# B&R Automation Studio project Panasonic_LinkaPowerCP2_A2021055 (part 45)

#### Main.st - Init, cyclic, exit code
```iecst
PROGRAM _INIT
	(* Insert code here *)
	SKTcpClientTrace_1.Params.IPportClient := 22000;
	SKTcpClientTrace_1.Cmd.LoggerOn:= FALSE;
END_PROGRAM

PROGRAM _CYCLIC

	//Priradenie indexu paletky//
    a:= P4_Etiketovacka.PAR.CisloPaletky;
	P4_Etiketovacka.PAR.CisloPaletky_STRING:= USINT_TO_STRING(a);

    //Parametre komunikácie//
    memcpy(ADR(SKTcpClientTrace_1.Params.IPaddrServ),ADR('192.168.128.250'),SIZEOF('192.168.128.250'));

    SKTcpClientTrace_1.Params.IPportServ := 12000;

	SKTcpClientTrace_1.pDevice := ADR('HDD_LOGGER');
	SKTcpClientTrace_1.pFile := ADR('logger_sktcpclienttrace_9.log');
    SKTcpClientTrace_1();

    //Parametre komunikácie//
    //Vstupy pre server//
    SKTcpClientTrace_1.Params.Packet.type := TRCB_P4_Etiketovacka_ST9.INPUTS.TYP_Prikazu;
    SKTcpClientTrace_1.Params.Packet.workplace := TRCB_P4_Etiketovacka_ST9.INPUTS.CisloStanice;
    SKTcpClientTrace_1.Params.Packet.rfid := TRCB_P4_Etiketovacka_ST9.INPUTS.CisloPaletky;
    SKTcpClientTrace_1.Params.Packet.master := TRCB_P4_Etiketovacka_ST9.INPUTS.QRkodPowerCP;
    SKTcpClientTrace_1.Params.Packet.dps1:= TRCB_P4_Etiketovacka_ST9.INPUTS.QRkodFiltra;
    SKTcpClientTrace_1.Params.Packet.dps2:= '';
    SKTcpClientTrace_1.Params.Packet.dps3:= '';
    SKTcpClientTrace_1.Params.Packet.dps4:= '';
    SKTcpClientTrace_1.Params.Packet.dps5:= '';
    SKTcpClientTrace_1.Params.Packet.operator_id := TRCB_P4_Etiketovacka_ST9.INPUTS.ID_Operatora;
    SKTcpClientTrace_1.Params.Packet.data_report:= TRCB_P4_Etiketovacka_ST9.INPUTS.Report;
    SKTcpClientTrace_1.Params.Packet.result := TRCB_P4_Etiketovacka_ST9.INPUTS.StavPaletky;

    //Výstupy zo servera//
    TRCB_P4_Etiketovacka_ST9.OUTPUTS.TYP_Prikazu:= SKTcpClientTrace_1.Internal.Splitter.out[1];
    TRCB_P4_Etiketovacka_ST9.OUTPUTS.CisloStanice:= SKTcpClientTrace_1.Internal.Splitter.out[2];
    TRCB_P4_Etiketovacka_ST9.OUTPUTS.CisloPaletky:= SKTcpClientTrace_1.Internal.Splitter.out[3];
    IF TRCB_P4_Etiketovacka_ST9.INPUTS.TYP_Prikazu = '0' THEN
        TRCB_P4_Etiketovacka_ST9.OUTPUTS.CisloEtikety:= SKTcpClientTrace_1.Internal.Splitter.out[4];
    ELSE
        TRCB_P4_Etiketovacka_ST9.OUTPUTS.QRkodPowerCP:= SKTcpClientTrace_1.Internal.Splitter.out[4];
    END_IF
    TRCB_P4_Etiketovacka_ST9.OUTPUTS.QRkodFiltra:= SKTcpClientTrace_1.Internal.Splitter.out[5];
    TRCB_P4_Etiketovacka_ST9.OUTPUTS.ID_Operatora:= SKTcpClientTrace_1.Internal.Splitter.out[10];
    TRCB_P4_Etiketovacka_ST9.OUTPUTS.DruhCinnostiNaPaletke:= SKTcpClientTrace_1.Internal.Splitter.out[11];
    TRCB_P4_Etiketovacka_ST9.OUTPUTS.PovolenieCinnostiNaPaletke:= SKTcpClientTrace_1.Internal.Splitter.out[12];

    //Volanie funkcie SequenceControl//
    SequenceControl(SC:= SC_KOM_Server);

    CASE SC_KOM_Server.Step OF

        0:
            SC_KOM_Server.StepName:= '0 - Nulovanie';
            SKTcpClientTrace_1.Cmd.Send:= FALSE;
            TRCB_P4_Etiketovacka_ST9.CMD.VyziadajStavPaletky_TYP1:= FALSE;
            TRCB_P4_Etiketovacka_ST9.CMD.PriradQRkodFiltra_TYP3:= FALSE;
            TRCB_P4_Etiketovacka_ST9.CMD.VyziadajCisloEtikety_TYP0:= FALSE;
			TRCB_P4_Etiketovacka_ST9.CMD.OdosliStavPaletky_TYP2:= FALSE;
			TRCB_P4_Etiketovacka_ST9.CMD.VyziadajStavPanatrace_TYP4:= FALSE;
            TRCB_P4_Etiketovacka_ST9.STATUS.KomunikaciaUkoncena:= FALSE;
			TRCB_P4_Etiketovacka_ST9.STATUS.KomunikaciaError:= FALSE;
			TRCB_P4_Etiketovacka_ST9.STATUS.KOM_READY:= FALSE;
            PocetDopytovNaServer:= 0;

            IF SKTcpClientTrace_1.Internal.Step = 0 THEN
                SKTcpClientTrace_1.Enable:= TRUE;
                SC_KOM_Server.ResetStep:= TRUE;
                SC_KOM_Server.Step:= 1;
            ELSIF SKTcpClientTrace_1.Internal.Step = 15 THEN
                SKTcpClientTrace_1.Enable:= TRUE;
                SC_KOM_Server.ResetStep:= TRUE;
                SC_KOM_Server.Step:= 1;
            ELSE
                SKTcpClientTrace_1.Enable:= FALSE;
            END_IF

        1:
            SC_KOM_Server.StepName:= '1 - Rozhodnutie o cinnosti';
            TRCB_P4_Etiketovacka_ST9.STATUS.KOM_READY:= TRUE;
			IF TRCB_P4_Etiketovacka_ST9.CMD.VyziadajStavPaletky_TYP1 THEN
                TRCB_P4_Etiketovacka_ST9.STATUS.KOM_READY:= FALSE;
				SC_KOM_Server.Step:= 10;
            ELSIF TRCB_P4_Etiketovacka_ST9.CMD.PriradQRkodFiltra_TYP3 THEN
                TRCB_P4_Etiketovacka_ST9.STATUS.KOM_READY:= FALSE;
				SC_KOM_Server.Step:= 20;
            ELSIF TRCB_P4_Etiketovacka_ST9.CMD.VyziadajCisloEtikety_TYP0 THEN
                TRCB_P4_Etiketovacka_ST9.STATUS.KOM_READY:= FALSE;
				SC_KOM_Server.Step:= 30;
            ELSIF TRCB_P4_Etiketovacka_ST9.CMD.OdosliStavPaletky_TYP2 THEN
				TRCB_P4_Etiketovacka_ST9.STATUS.KOM_READY:= FALSE;
				SC_KOM_Server.Step:= 40;
			ELSIF TRCB_P4_Etiketovacka_ST9.CMD.VyziadajStavPanatrace_TYP4 THEN
				TRCB_P4_Etiketovacka_ST9.STATUS.KOM_READY:= FALSE;
				SC_KOM_Server.Step:= 50;
            END_IF

        10:
            SC_KOM_Server.StepName:= '10 - Vyziadanie stavu paletky - odoslanie dat na server';
            SC_KOM_Server.IdleTime.PT:= T#3s;
            SC_KOM_Server.AlarmTime.PT:= T#10s;
            SC_KOM_Server.AlarmTime.IN:= TRUE;

			TRCB_P4_Etiketovacka_ST9.INPUTS.CisloPaletky:= 'Pal';
			brsstrcat(ADR(TRCB_P4_Etiketovacka_ST9.INPUTS.CisloPaletky), ADR(P4_Etiketovacka.PAR.CisloPaletky_STRING));

            TRCB_P4_Etiketovacka_ST9.INPUTS.TYP_Prikazu:= '1';
            TRCB_P4_Etiketovacka_ST9.INPUTS.CisloStanice:= 'ST9';
            TRCB_P4_Etiketovacka_ST9.INPUTS.QRkodPowerCP:= Paletka[a].PAR.QRkodPowerCP;
            TRCB_P4_Etiketovacka_ST9.INPUTS.QRkodFiltra:= '';
            TRCB_P4_Etiketovacka_ST9.INPUTS.ID_Operatora:= Paletka[a].PAR.ID_Operatora;
            TRCB_P4_Etiketovacka_ST9.INPUTS.Report:= '';
            TRCB_P4_Etiketovacka_ST9.INPUTS.StavPaletky:= 'OK';

			IF SKTcpClientTrace_1.Status.staReadyToSend AND NOT SKTcpClientTrace_1.Cmd.Close THEN
				TRCB_P4_Etiketovacka_ST9.OUTPUTS.TYP_Prikazu:= '';
				SKTcpClientTrace_1.Cmd.Send:= TRUE;
				SC_KOM_Server.ResetStep:= TRUE;
				SC_KOM_Server.Step:= 13;
			END_IF

		13:
            SC_KOM_Server.StepName:= '13 - Vyziadanie stavu paletky - odpoved servera';
            SC_KOM_Server.IdleTime.PT:= T#3s;
            SC_KOM_Server.AlarmTime.PT:= T#7s;
            SC_KOM_Server.AlarmTime.IN:= TRUE;

            IF SKTcpClientTrace_1.Status.staReceived AND
                (TRCB_P4_Etiketovacka_ST9.OUTPUTS.TYP_Prikazu = TRCB_P4_Etiketovacka_ST9.INPUTS.TYP_Prikazu) AND
                (TRCB_P4_Etiketovacka_ST9.OUTPUTS.QRkodPowerCP = TRCB_P4_Etiketovacka_ST9.INPUTS.QRkodPowerCP) THEN
                TRCB_P4_Etiketovacka_ST9.STATUS.KomunikaciaUkoncena:= TRUE;
                SC_KOM_Server.ResetStep:= TRUE;
                SC_KOM_Server.Step:= 15;
            ELSIF SC_KOM_Server.AlarmTime.Q AND NOT SKTcpClientTrace_1.Status.staSending THEN
                PocetDopytovNaServer:= PocetDopytovNaServer + 1;
				SKTcpClientTrace_1.Cmd.Send:= FALSE;
				SKTcpClientTrace_1.Cmd.Close:= TRUE;
				SC_KOM_Server.ResetStep:= TRUE;
                SC_KOM_Server.Step:= 14;
            END_IF

        14:
            SC_KOM_Server.StepName:= '14 - Vyziadanie stavu paletky - cakam na opatovny dopyt na server';
            SC_KOM_Server.IdleTime.PT:= T#1s;
            SC_KOM_Server.AlarmTime.PT:= T#10s;
            SC_KOM_Server.IdleTime.IN:= TRUE;

            IF PocetDopytovNaServer < 3 THEN
                IF SC_KOM_Server.IdleTime.Q THEN
                    SC_KOM_Server.ResetStep:= TRUE;
                    SC_KOM_Server.Step:= 10;
                END_IF
            ELSE
                TRCB_P4_Etiketovacka_ST9.STATUS.KomunikaciaError:= TRUE;
                SC_KOM_Server.ResetStep:= TRUE;
                SC_KOM_Server.Step:= 15;
            END_IF

        15:
            SC_KOM_Server.StepName:= '15 - Vyziadanie stavu paletky - cakam na ukoncenie komunikacie';
            SC_KOM_Server.IdleTime.PT:= T#3s;
            SC_KOM_Server.AlarmTime.PT:= T#10s;

            IF NOT TRCB_P4_Etiketovacka_ST9.CMD.VyziadajStavPaletky_TYP1 THEN
                SC_KOM_Server.ResetStep:= TRUE;
                SC_KOM_Server.Step:= 0;
            END_IF

        20:
            SC_KOM_Server.StepName:= '20 - Priradenie QR kodu - odoslanie dat na server';
            SC_KOM_Server.IdleTime.PT:= T#3s;
            SC_KOM_Server.AlarmTime.PT:= T#10s;

            TRCB_P4_Etiketovacka_ST9.INPUTS.TYP_Prikazu:= '3';
            TRCB_P4_Etiketovacka_ST9.INPUTS.CisloStanice:= 'ST9';
            TRCB_P4_Etiketovacka_ST9.INPUTS.CisloPaletky;
            TRCB_P4_Etiketovacka_ST9.INPUTS.QRkodPowerCP:= Paletka[a].PAR.QRkodPowerCP;
            TRCB_P4_Etiketovacka_ST9.INPUTS.QRkodFiltra:= '';
            TRCB_P4_Etiketovacka_ST9.INPUTS.ID_Operatora:= Paletka[a].PAR.ID_Operatora;
            TRCB_P4_Etiketovacka_ST9.INPUTS.Report:= '';
            TRCB_P4_Etiketovacka_ST9.INPUTS.StavPaletky:= 'OK';
            SKTcpClientTrace_1.Cmd.Send:= TRUE;

            IF SKTcpClientTrace_1.Cmd.Send AND NOT SKTcpClientTrace_1.Status.staReceived AND NOT SKTcpClientTrace_1.Status.staError THEN
                SC_KOM_Server.ResetStep:= TRUE;
                SC_KOM_Server.Step:= 23;
            END_IF

        23:
            SC_KOM_Server.StepName:= '23 - Priradenie QR kodu - odpoved servera';
            SC_KOM_Server.IdleTime.PT:= T#3s;
            SC_KOM_Server.AlarmTime.PT:= T#20s;
            SC_KOM_Server.AlarmTime.IN:= TRUE;

            IF SKTcpClientTrace_1.Status.staReceived AND
                (TRCB_P4_Etiketovacka_ST9.OUTPUTS.TYP_Prikazu = TRCB_P4_Etiketovacka_ST9.INPUTS.TYP_Prikazu) AND
                (TRCB_P4_Etiketovacka_ST9.OUTPUTS.QRkodPowerCP = TRCB_P4_Etiketovacka_ST9.INPUTS.QRkodPowerCP) THEN
                TRCB_P4_Etiketovacka_ST9.STATUS.KomunikaciaUkoncena:= TRUE;
                SC_KOM_Server.ResetStep:= TRUE;
                SC_KOM_Server.Step:= 25;
            ELSIF SC_KOM_Server.AlarmTime.Q THEN
                TRCB_P4_Etiketovacka_ST9.STATUS.KomunikaciaError:= TRUE;
                SC_KOM_Server.ResetStep:= TRUE;
                SC_KOM_Server.Step:= 25;
            END_IF

        25:
            SC_KOM_Server.StepName:= '25 - Priradenie QR kodu - cakam na ukoncenie komunikacie';
            SC_KOM_Server.IdleTime.PT:= T#3s;
            SC_KOM_Server.AlarmTime.PT:= T#10s;

            IF NOT TRCB_P4_Etiketovacka_ST9.CMD.PriradQRkodFiltra_TYP3 THEN
                SC_KOM_Server.ResetStep:= TRUE;
                SC_KOM_Server.Step:= 0;
            END_IF

        30:
            SC_KOM_Server.StepName:= '30 - Vyziadanie serioveho cisla - odoslanie dat na server';
            SC_KOM_Server.IdleTime.PT:= T#3s;
            SC_KOM_Server.AlarmTime.PT:= T#20s;
            SC_KOM_Server.AlarmTime.IN:= TRUE;

			TRCB_P4_Etiketovacka_ST9.INPUTS.CisloPaletky:= 'Pal';
			brsstrcat(ADR(TRCB_P4_Etiketovacka_ST9.INPUTS.CisloPaletky), ADR(P4_Etiketovacka.PAR.CisloPaletky_STRING));

            TRCB_P4_Etiketovacka_ST9.INPUTS.TYP_Prikazu:= '0';
            TRCB_P4_Etiketovacka_ST9.INPUTS.CisloStanice:= 'ST9';
            TRCB_P4_Etiketovacka_ST9.INPUTS.QRkodPowerCP:= '';
            TRCB_P4_Etiketovacka_ST9.INPUTS.QRkodFiltra:= '';
            TRCB_P4_Etiketovacka_ST9.INPUTS.ID_Operatora:= Paletka[a].PAR.ID_Operatora;
            TRCB_P4_Etiketovacka_ST9.INPUTS.Report:= '';
            TRCB_P4_Etiketovacka_ST9.INPUTS.StavPaletky:= 'OK';

			IF SKTcpClientTrace_1.Status.staReadyToSend AND NOT SKTcpClientTrace_1.Cmd.Close THEN
				TRCB_P4_Etiketovacka_ST9.OUTPUTS.TYP_Prikazu:= '';
				SKTcpClientTrace_1.Cmd.Send:= TRUE;
				SC_KOM_Server.ResetStep:= TRUE;
				SC_KOM_Server.Step:= 33;
			END_IF

        33:
            SC_KOM_Server.StepName:= '33 - Vyziadanie serioveho cisla - odpoved servera';
			SC_KOM_Server.IdleTime.PT:= T#3s;
            SC_KOM_Server.AlarmTime.PT:= T#7s;
            SC_KOM_Server.AlarmTime.IN:= TRUE;

            IF SKTcpClientTrace_1.Status.staReceived AND
                (TRCB_P4_Etiketovacka_ST9.OUTPUTS.TYP_Prikazu = TRCB_P4_Etiketovacka_ST9.INPUTS.TYP_Prikazu) THEN
                TRCB_P4_Etiketovacka_ST9.STATUS.KomunikaciaUkoncena:= TRUE;
                SC_KOM_Server.ResetStep:= TRUE;
                SC_KOM_Server.Step:= 35;
            ELSIF SC_KOM_Server.AlarmTime.Q AND NOT SKTcpClientTrace_1.Status.staSending THEN
                PocetDopytovNaServer:= PocetDopytovNaServer + 1;
				SKTcpClientTrace_1.Cmd.Send:= FALSE;
				SKTcpClientTrace_1.Cmd.Close:= TRUE;
				SC_KOM_Server.ResetStep:= TRUE;
                SC_KOM_Server.Step:= 34;
            END_IF

        34:
            SC_KOM_Server.StepName:= '34 - Vyziadanie serioveho cisla - cakam na opatovny dopyt na server';
            SC_KOM_Server.IdleTime.PT:= T#1s;
            SC_KOM_Server.AlarmTime.PT:= T#10s;
            SC_KOM_Server.IdleTime.IN:= TRUE;
            SKTcpClientTrace_1.Cmd.Send:= FALSE;

            IF PocetDopytovNaServer < 3 THEN
                IF SC_KOM_Server.IdleTime.Q THEN
                    SC_KOM_Server.ResetStep:= TRUE;
                    SC_KOM_Server.Step:= 30;
                END_IF
            ELSE
                TRCB_P4_Etiketovacka_ST9.STATUS.KomunikaciaError:= TRUE;
                SC_KOM_Server.ResetStep:= TRUE;
                SC_KOM_Server.Step:= 35;
            END_IF

        35:
            SC_KOM_Server.StepName:= '35 - Vyziadanie serioveho cisla - cakam na ukoncenie komunikacie';
            SC_KOM_Server.IdleTime.PT:= T#3s;
            SC_KOM_Server.AlarmTime.PT:= T#10s;

            IF NOT TRCB_P4_Etiketovacka_ST9.CMD.VyziadajCisloEtikety_TYP0 THEN
                SC_KOM_Server.ResetStep:= TRUE;
                SC_KOM_Server.Step:= 0;
            END_IF

        40:
            SC_KOM_Server.StepName:= '40 - Odoslanie stavu paletky - odoslanie dat na server';
            SC_KOM_Server.IdleTime.PT:= T#3s;
            SC_KOM_Server.AlarmTime.PT:= T#20s;
            SC_KOM_Server.AlarmTime.IN:= TRUE;

            IF NOT SC_KOM_Server.Switch1 THEN
                brsmemset(ADR(Report),0,SIZEOF(Report));
               	brsmemset(ADR(TRCB_P4_Etiketovacka_ST9.INPUTS.Report), 0, SIZEOF(TRCB_P4_Etiketovacka_ST9.INPUTS.Report));

				//Kamera 15//
                Report[0].PoradoveCislo:= '1';
                Report[0].Popis:= 'KAM_15_KontrolaEtikety';
                Report[0].FormatHodnoty:= '2';
                Report[0].Tolerancia_MIN_Hodnota:= '';
                Report[0].Tolerancia_MAX_Hodnota:= '';
                Report[0].Nominal:= 'OK';
                Report[0].Tolerancia_MIN_Jednotky:= '';
                Report[0].Tolerancia_MAX_Jednotky:= '';
                IF Reports.Kamery.P4_CAM15_KontrolaPaletky = 'PASS' THEN
                    Report[0].NameranaHodnota:= 'OK';
                ELSE
                    Report[0].NameranaHodnota:= 'NG';
                END_IF
                Report[0].NameranaHodnota_Jednotky:= '';
                Report[0].VyslednyResult:= Reports.Kamery.P4_CAM15_KontrolaPaletky;
                SKTcpClientNewCsvEntry(Report[0].PoradoveCislo,Report[0].Popis,Report[0].FormatHodnoty,Report[0].Tolerancia_MIN_Hodnota,Report[0].Tolerancia_MAX_Hodnota,Report[0].Nominal,Report[0].Tolerancia_MIN_Jednotky,Report[0].Tolerancia_MAX_Jednotky,Report[0].NameranaHodnota,Report[0].NameranaHodnota_Jednotky,Report[0].VyslednyResult, ADR(TRCB_P4_Etiketovacka_ST9.INPUTS.Report));
                SC_KOM_Server.Switch1:= TRUE;
            END_IF

			TRCB_P4_Etiketovacka_ST9.INPUTS.CisloPaletky:= 'Pal';
			brsstrcat(ADR(TRCB_P4_Etiketovacka_ST9.INPUTS.CisloPaletky), ADR(P4_Etiketovacka.PAR.CisloPaletky_STRING));

            TRCB_P4_Etiketovacka_ST9.INPUTS.TYP_Prikazu:= '2';
            TRCB_P4_Etiketovacka_ST9.INPUTS.CisloStanice:= 'ST9';
            TRCB_P4_Etiketovacka_ST9.INPUTS.QRkodPowerCP:= Paletka[a].PAR.QRkodPowerCP;
            TRCB_P4_Etiketovacka_ST9.INPUTS.QRkodFiltra:= '';
            TRCB_P4_Etiketovacka_ST9.INPUTS.ID_Operatora:= Paletka[a].PAR.ID_Operatora;
            TRCB_P4_Etiketovacka_ST9.INPUTS.StavPaletky:= Paletka[a].PAR.StavPowerCP;

			IF SKTcpClientTrace_1.Status.staReadyToSend AND NOT SKTcpClientTrace_1.Cmd.Close THEN
				TRCB_P4_Etiketovacka_ST9.OUTPUTS.TYP_Prikazu:= '';
				SKTcpClientTrace_1.Cmd.Send:= TRUE;
				SC_KOM_Server.ResetStep:= TRUE;
				SC_KOM_Server.Step:= 43;
			END_IF

        43:
            SC_KOM_Server.StepName:= '43 - Odoslanie stavu paletky - odpoved servera';
			SC_KOM_Server.IdleTime.PT:= T#3s;
            SC_KOM_Server.AlarmTime.PT:= T#7s;
            SC_KOM_Server.AlarmTime.IN:= TRUE;

            IF SKTcpClientTrace_1.Status.staReceived AND
                (TRCB_P4_Etiketovacka_ST9.OUTPUTS.TYP_Prikazu = TRCB_P4_Etiketovacka_ST9.INPUTS.TYP_Prikazu) AND
                (TRCB_P4_Etiketovacka_ST9.OUTPUTS.QRkodPowerCP = TRCB_P4_Etiketovacka_ST9.INPUTS.QRkodPowerCP) THEN
                TRCB_P4_Etiketovacka_ST9.STATUS.KomunikaciaUkoncena:= TRUE;
                SC_KOM_Server.ResetStep:= TRUE;
                SC_KOM_Server.Step:= 45;
            ELSIF SC_KOM_Server.AlarmTime.Q AND NOT SKTcpClientTrace_1.Status.staSending THEN
                PocetDopytovNaServer:= PocetDopytovNaServer + 1;
				SKTcpClientTrace_1.Cmd.Send:= FALSE;
				SKTcpClientTrace_1.Cmd.Close:= TRUE;
				SC_KOM_Server.ResetStep:= TRUE;
                SC_KOM_Server.Step:= 44;
            END_IF

        44:
            SC_KOM_Server.StepName:= '44 - Odoslanie stavu paletky - cakam na opatovny dopyt na server';
            SC_KOM_Server.IdleTime.PT:= T#1s;
            SC_KOM_Server.AlarmTime.PT:= T#10s;
            SC_KOM_Server.IdleTime.IN:= TRUE;
            SKTcpClientTrace_1.Cmd.Send:= FALSE;

            IF PocetDopytovNaServer < 3 THEN
                IF SC_KOM_Server.IdleTime.Q THEN
                    SC_KOM_Server.ResetStep:= TRUE;
                    SC_KOM_Server.Step:= 40;
                END_IF
            ELSE
                TRCB_P4_Etiketovacka_ST9.STATUS.KomunikaciaError:= TRUE;
                SC_KOM_Server.ResetStep:= TRUE;
                SC_KOM_Server.Step:= 45;
            END_IF

        45:
            SC_KOM_Server.StepName:= '45 - Odoslanie stavu paletky - cakam na ukoncenie komunikacie';
            SC_KOM_Server.IdleTime.PT:= T#3s;
            SC_KOM_Server.AlarmTime.PT:= T#10s;

            IF NOT TRCB_P4_Etiketovacka_ST9.CMD.OdosliStavPaletky_TYP2 THEN
                SC_KOM_Server.ResetStep:= TRUE;
                SC_KOM_Server.Step:= 0;
            END_IF

		50:
			SC_KOM_Server.StepName:= '50 - Vyziadanie stavu Panatrace - odoslanie dat na server';
			SC_KOM_Server.IdleTime.PT:= T#3s;
			SC_KOM_Server.AlarmTime.PT:= T#10s;
			SC_KOM_Server.AlarmTime.IN:= TRUE;

			TRCB_P4_Etiketovacka_ST9.INPUTS.TYP_Prikazu:= '4';
			TRCB_P4_Etiketovacka_ST9.INPUTS.CisloStanice:= 'ST9';
			TRCB_P4_Etiketovacka_ST9.INPUTS.CisloPaletky:= '';
			TRCB_P4_Etiketovacka_ST9.INPUTS.QRkodPowerCP:= '';
			TRCB_P4_Etiketovacka_ST9.INPUTS.QRkodFiltra:= '';
			TRCB_P4_Etiketovacka_ST9.INPUTS.ID_Operatora:= '';
			TRCB_P4_Etiketovacka_ST9.INPUTS.Report:= '';
			TRCB_P4_Etiketovacka_ST9.INPUTS.StavPaletky:= '';

			IF SKTcpClientTrace_1.Status.staReadyToSend AND NOT SKTcpClientTrace_1.Cmd.Close THEN
				TRCB_P4_Etiketovacka_ST9.OUTPUTS.TYP_Prikazu:= '';
				SKTcpClientTrace_1.Cmd.Send:= TRUE;
				SC_KOM_Server.ResetStep:= TRUE;
				SC_KOM_Server.Step:= 53;
			END_IF

		53:
			SC_KOM_Server.StepName:= '53 - Vyziadanie stavu paletky - odpoved servera';
			SC_KOM_Server.IdleTime.PT:= T#30s;
			SC_KOM_Server.AlarmTime.PT:= T#7s;
			SC_KOM_Server.AlarmTime.IN:= TRUE;

			IF SKTcpClientTrace_1.Status.staReceived AND TRCB_P4_Etiketovacka_ST9.OUTPUTS.TYP_Prikazu = TRCB_P4_Etiketovacka_ST9.INPUTS.TYP_Prikazu THEN
				TRCB_P4_Etiketovacka_ST9.STATUS.KomunikaciaUkoncena:= TRUE;
				SC_KOM_Server.ResetStep:= TRUE;
				SC_KOM_Server.Step:= 55;
			ELSIF SC_KOM_Server.AlarmTime.Q AND NOT SKTcpClientTrace_1.Status.staSending THEN
				PocetDopytovNaServer:= PocetDopytovNaServer + 1;
				SKTcpClientTrace_1.Cmd.Send:= FALSE;
				SKTcpClientTrace_1.Cmd.Close:= TRUE;
				SC_KOM_Server.ResetStep:= TRUE;
				SC_KOM_Server.Step:= 54;
			END_IF

		54:
			SC_KOM_Server.StepName:= '54 - Vyziadanie stavu paletky - cakam na opatovny dopyt na server';
			SC_KOM_Server.IdleTime.PT:= T#1s;
			SC_KOM_Server.AlarmTime.PT:= T#10s;
			SC_KOM_Server.IdleTime.IN:= TRUE;

			IF PocetDopytovNaServer < 3 THEN
				IF SC_KOM_Server.IdleTime.Q THEN
					SC_KOM_Server.ResetStep:= TRUE;
					SC_KOM_Server.Step:= 50;
				END_IF
			ELSE
				TRCB_P4_Etiketovacka_ST9.STATUS.KomunikaciaError:= TRUE;
				SC_KOM_Server.ResetStep:= TRUE;
				SC_KOM_Server.Step:= 55;
			END_IF

		55:
			SC_KOM_Server.StepName:= '55 - Vyziadanie stavu paletky - cakam na ukoncenie komunikacie';
			SC_KOM_Server.IdleTime.PT:= T#3s;
			SC_KOM_Server.AlarmTime.PT:= T#10s;

			IF NOT TRCB_P4_Etiketovacka_ST9.CMD.VyziadajStavPanatrace_TYP4 THEN
				SC_KOM_Server.ResetStep:= TRUE;
				SC_KOM_Server.Step:= 0;
			END_IF

    END_CASE

END_PROGRAM

PROGRAM _EXIT
	(* Insert code here *)

END_PROGRAM
```

#### Types.typ - Local data types
```iecst
TYPE
	Report_typ : 	STRUCT
		PoradoveCislo : STRING[2]; (*IDstep - Poradové čislo reportu*)
		Popis : STRING[100]; (*Description - Popis*)
		FormatHodnoty : STRING[2]; (*TypValue - Format zaslané hodnoty  1- Číslo, 2 - Znak*)
		Tolerancia_MIN_Hodnota : STRING[10]; (*MinTol - Minimálna tolerancia meranej veličiny*)
		Tolerancia_MAX_Hodnota : STRING[10]; (*MaxTol - Maximálna tolerancia meranej veličiny*)
		Nominal : STRING[10]; (*Nom - Ak jezvolený formát string tak tu zadáme OK inak je prazdna*)
		Tolerancia_MIN_Jednotky : STRING[10]; (*MinEle - Jednotky minimálnej tolerancie veličiny*)
		Tolerancia_MAX_Jednotky : STRING[10]; (*MaxEle - Jednotky maximálnej tolerancie veličiny*)
		NameranaHodnota : STRING[10]; (*Value - Namerana hodnota veličiny, ak su kamery tak bude hodnota OK alebo NG*)
		NameranaHodnota_Jednotky : STRING[10]; (*ValEle - Jednotky nameranej veličiny*)
		VyslednyResult : STRING[5]; (*Result - Výsledný result  PASS, FAIL, SKIP*)
	END_STRUCT;
END_TYPE
```

#### Variables.var - Local variables
```iecst
VAR
	SC_KOM_Server : SequenceControlTyp;
	SKTcpClientTrace_1 : SKTcpClientTrace;
	a : USINT;
	Report : ARRAY[0..50] OF Report_typ;
	PocetDopytovNaServer : USINT;
END_VAR
```

### Program Logical/TracebilitySystem/P4_Vytah_ST10 (IEC)

#### Main.st - Init, cyclic, exit code
```iecst
PROGRAM _INIT
	(* Insert code here *)
	SKTcpClientTrace_1.Params.IPportClient := 23000;
	SKTcpClientTrace_1.Cmd.LoggerOn:= FALSE;
END_PROGRAM

PROGRAM _CYCLIC

	//Priradenie indexu paletky//
    a:= P4_Vytah.PAR.CisloPaletky;
	P4_Vytah.PAR.CisloPaletky_STRING:= USINT_TO_STRING(a);

    //Parametre komunikácie//
    memcpy(ADR(SKTcpClientTrace_1.Params.IPaddrServ),ADR('192.168.128.250'),SIZEOF('192.168.128.250'));

    SKTcpClientTrace_1.Params.IPportServ := 12000;

	SKTcpClientTrace_1.pDevice := ADR('HDD_LOGGER');
	SKTcpClientTrace_1.pFile := ADR('logger_sktcpclienttrace_10.log');
    SKTcpClientTrace_1();

    //Parametre komunikácie//
    //Vstupy pre server//
    SKTcpClientTrace_1.Params.Packet.type := TRCB_P4_Vytah_ST10.INPUTS.TYP_Prikazu;
    SKTcpClientTrace_1.Params.Packet.workplace := TRCB_P4_Vytah_ST10.INPUTS.CisloStanice;
    SKTcpClientTrace_1.Params.Packet.rfid := TRCB_P4_Vytah_ST10.INPUTS.CisloPaletky;
    SKTcpClientTrace_1.Params.Packet.master := TRCB_P4_Vytah_ST10.INPUTS.QRkodPowerCP;
    SKTcpClientTrace_1.Params.Packet.dps1:= TRCB_P4_Vytah_ST10.INPUTS.QRkodFiltra;
    SKTcpClientTrace_1.Params.Packet.dps2:= '';
    SKTcpClientTrace_1.Params.Packet.dps3:= '';
    SKTcpClientTrace_1.Params.Packet.dps4:= '';
    SKTcpClientTrace_1.Params.Packet.dps5:= '';
    SKTcpClientTrace_1.Params.Packet.operator_id := TRCB_P4_Vytah_ST10.INPUTS.ID_Operatora;
    SKTcpClientTrace_1.Params.Packet.data_report:= TRCB_P4_Vytah_ST10.INPUTS.Report;
    SKTcpClientTrace_1.Params.Packet.result := TRCB_P4_Vytah_ST10.INPUTS.StavPaletky;

    //Výstupy zo servera//
    TRCB_P4_Vytah_ST10.OUTPUTS.TYP_Prikazu:= SKTcpClientTrace_1.Internal.Splitter.out[1];
    TRCB_P4_Vytah_ST10.OUTPUTS.CisloStanice:= SKTcpClientTrace_1.Internal.Splitter.out[2];
    TRCB_P4_Vytah_ST10.OUTPUTS.CisloPaletky:= SKTcpClientTrace_1.Internal.Splitter.out[3];
    IF TRCB_P4_Vytah_ST10.INPUTS.TYP_Prikazu = '0' THEN
        TRCB_P4_Vytah_ST10.OUTPUTS.CisloEtikety:= SKTcpClientTrace_1.Internal.Splitter.out[4];
    ELSE
        TRCB_P4_Vytah_ST10.OUTPUTS.QRkodPowerCP:= SKTcpClientTrace_1.Internal.Splitter.out[4];
    END_IF
    TRCB_P4_Vytah_ST10.OUTPUTS.QRkodFiltra:= SKTcpClientTrace_1.Internal.Splitter.out[5];
    TRCB_P4_Vytah_ST10.OUTPUTS.ID_Operatora:= SKTcpClientTrace_1.Internal.Splitter.out[10];
    TRCB_P4_Vytah_ST10.OUTPUTS.DruhCinnostiNaPaletke:= SKTcpClientTrace_1.Internal.Splitter.out[11];
    TRCB_P4_Vytah_ST10.OUTPUTS.PovolenieCinnostiNaPaletke:= SKTcpClientTrace_1.Internal.Splitter.out[12];

    //Volanie funkcie SequenceControl//
    SequenceControl(SC:= SC_KOM_Server);

    CASE SC_KOM_Server.Step OF

        0:
            SC_KOM_Server.StepName:= '0 - Nulovanie';
            SKTcpClientTrace_1.Cmd.Send:= FALSE;
            TRCB_P4_Vytah_ST10.CMD.VyziadajStavPaletky_TYP1:= FALSE;
            TRCB_P4_Vytah_ST10.CMD.PriradQRkodFiltra_TYP3:= FALSE;
            TRCB_P4_Vytah_ST10.CMD.VyziadajCisloEtikety_TYP0:= FALSE;
			TRCB_P4_Vytah_ST10.CMD.OdosliStavPaletky_TYP2:= FALSE;
			TRCB_P4_Vytah_ST10.CMD.VyziadajStavPanatrace_TYP4:= FALSE;
            TRCB_P4_Vytah_ST10.STATUS.KomunikaciaUkoncena:= FALSE;
			TRCB_P4_Vytah_ST10.STATUS.KomunikaciaError:= FALSE;
			TRCB_P4_Vytah_ST10.STATUS.KOM_READY:= FALSE;
            PocetDopytovNaServer:= 0;

            IF SKTcpClientTrace_1.Internal.Step = 0 THEN
                SKTcpClientTrace_1.Enable:= TRUE;
                SC_KOM_Server.ResetStep:= TRUE;
                SC_KOM_Server.Step:= 1;
            ELSIF SKTcpClientTrace_1.Internal.Step = 15 THEN
                SKTcpClientTrace_1.Enable:= TRUE;
                SC_KOM_Server.ResetStep:= TRUE;
                SC_KOM_Server.Step:= 1;
            ELSE
                SKTcpClientTrace_1.Enable:= FALSE;
            END_IF

        1:
            SC_KOM_Server.StepName:= '1 - Rozhodnutie o cinnosti';
            TRCB_P4_Vytah_ST10.STATUS.KOM_READY:= TRUE;
			IF TRCB_P4_Vytah_ST10.CMD.VyziadajStavPaletky_TYP1 THEN
                TRCB_P4_Vytah_ST10.STATUS.KOM_READY:= FALSE;
				SC_KOM_Server.Step:= 10;
            ELSIF TRCB_P4_Vytah_ST10.CMD.PriradQRkodFiltra_TYP3 THEN
                TRCB_P4_Vytah_ST10.STATUS.KOM_READY:= FALSE;
				SC_KOM_Server.Step:= 20;
            ELSIF TRCB_P4_Vytah_ST10.CMD.VyziadajCisloEtikety_TYP0 THEN
                TRCB_P4_Vytah_ST10.STATUS.KOM_READY:= FALSE;
				SC_KOM_Server.Step:= 30;
            ELSIF TRCB_P4_Vytah_ST10.CMD.OdosliStavPaletky_TYP2 THEN
				TRCB_P4_Vytah_ST10.STATUS.KOM_READY:= FALSE;
				SC_KOM_Server.Step:= 40;
			ELSIF TRCB_P4_Vytah_ST10.CMD.VyziadajStavPanatrace_TYP4 THEN
				TRCB_P4_Vytah_ST10.STATUS.KOM_READY:= FALSE;
				SC_KOM_Server.Step:= 50;
            END_IF

        10:
            SC_KOM_Server.StepName:= '10 - Vyziadanie stavu paletky - odoslanie dat na server';
            SC_KOM_Server.IdleTime.PT:= T#3s;
            SC_KOM_Server.AlarmTime.PT:= T#10s;
            SC_KOM_Server.AlarmTime.IN:= TRUE;

			TRCB_P4_Vytah_ST10.INPUTS.CisloPaletky:= 'Pal';
			brsstrcat(ADR(TRCB_P4_Vytah_ST10.INPUTS.CisloPaletky), ADR(P4_Vytah.PAR.CisloPaletky_STRING));

            TRCB_P4_Vytah_ST10.INPUTS.TYP_Prikazu:= '1';
            TRCB_P4_Vytah_ST10.INPUTS.CisloStanice:= 'ST10';
            TRCB_P4_Vytah_ST10.INPUTS.QRkodPowerCP:= Paletka[a].PAR.QRkodPowerCP;
            TRCB_P4_Vytah_ST10.INPUTS.QRkodFiltra:= '';
            TRCB_P4_Vytah_ST10.INPUTS.ID_Operatora:= Paletka[a].PAR.ID_Operatora;
            TRCB_P4_Vytah_ST10.INPUTS.Report:= '';
            TRCB_P4_Vytah_ST10.INPUTS.StavPaletky:= 'OK';

			IF SKTcpClientTrace_1.Status.staReadyToSend AND NOT SKTcpClientTrace_1.Cmd.Close THEN
				TRCB_P4_Vytah_ST10.OUTPUTS.TYP_Prikazu:= '';
				SKTcpClientTrace_1.Cmd.Send:= TRUE;
				SC_KOM_Server.ResetStep:= TRUE;
				SC_KOM_Server.Step:= 13;
			END_IF

		13:
            SC_KOM_Server.StepName:= '13 - Vyziadanie stavu paletky - odpoved servera';
            SC_KOM_Server.IdleTime.PT:= T#3s;
            SC_KOM_Server.AlarmTime.PT:= T#7s;
            SC_KOM_Server.AlarmTime.IN:= TRUE;

            IF SKTcpClientTrace_1.Status.staReceived AND
                (TRCB_P4_Vytah_ST10.OUTPUTS.TYP_Prikazu = TRCB_P4_Vytah_ST10.INPUTS.TYP_Prikazu) AND
                (TRCB_P4_Vytah_ST10.OUTPUTS.QRkodPowerCP = TRCB_P4_Vytah_ST10.INPUTS.QRkodPowerCP) THEN
                TRCB_P4_Vytah_ST10.STATUS.KomunikaciaUkoncena:= TRUE;
                SC_KOM_Server.ResetStep:= TRUE;
                SC_KOM_Server.Step:= 15;
            ELSIF SC_KOM_Server.AlarmTime.Q AND NOT SKTcpClientTrace_1.Status.staSending THEN
                PocetDopytovNaServer:= PocetDopytovNaServer + 1;
				SKTcpClientTrace_1.Cmd.Send:= FALSE;
				SKTcpClientTrace_1.Cmd.Close:= TRUE;
				SC_KOM_Server.ResetStep:= TRUE;
                SC_KOM_Server.Step:= 14;
            END_IF

        14:
            SC_KOM_Server.StepName:= '14 - Vyziadanie stavu paletky - cakam na opatovny dopyt na server';
            SC_KOM_Server.IdleTime.PT:= T#1s;
            SC_KOM_Server.AlarmTime.PT:= T#10s;
            SC_KOM_Server.IdleTime.IN:= TRUE;

            IF PocetDopytovNaServer < 3 THEN
                IF SC_KOM_Server.IdleTime.Q THEN
                    SC_KOM_Server.ResetStep:= TRUE;
                    SC_KOM_Server.Step:= 10;
                END_IF
            ELSE
                TRCB_P4_Vytah_ST10.STATUS.KomunikaciaError:= TRUE;
                SC_KOM_Server.ResetStep:= TRUE;
                SC_KOM_Server.Step:= 15;
            END_IF

        15:
            SC_KOM_Server.StepName:= '15 - Vyziadanie stavu paletky - cakam na ukoncenie komunikacie';
            SC_KOM_Server.IdleTime.PT:= T#3s;
            SC_KOM_Server.AlarmTime.PT:= T#10s;

            IF NOT TRCB_P4_Vytah_ST10.CMD.VyziadajStavPaletky_TYP1 THEN
                SC_KOM_Server.ResetStep:= TRUE;
                SC_KOM_Server.Step:= 0;
            END_IF

        20:
            SC_KOM_Server.StepName:= '20 - Priradenie QR kodu - odoslanie dat na server';
            SC_KOM_Server.IdleTime.PT:= T#3s;
            SC_KOM_Server.AlarmTime.PT:= T#10s;

            TRCB_P4_Vytah_ST10.INPUTS.TYP_Prikazu:= '3';
            TRCB_P4_Vytah_ST10.INPUTS.CisloStanice:= 'ST10';
            TRCB_P4_Vytah_ST10.INPUTS.CisloPaletky;
            TRCB_P4_Vytah_ST10.INPUTS.QRkodPowerCP:= Paletka[a].PAR.QRkodPowerCP;
            TRCB_P4_Vytah_ST10.INPUTS.QRkodFiltra:= Paletka[a].PAR.QRkodFiltra_4F5F;
            TRCB_P4_Vytah_ST10.INPUTS.ID_Operatora:= Paletka[a].PAR.ID_Operatora;
            TRCB_P4_Vytah_ST10.INPUTS.Report:= '';
            TRCB_P4_Vytah_ST10.INPUTS.StavPaletky:= 'OK';
            SKTcpClientTrace_1.Cmd.Send:= TRUE;

            IF SKTcpClientTrace_1.Cmd.Send AND NOT SKTcpClientTrace_1.Status.staReceived AND NOT SKTcpClientTrace_1.Status.staError THEN
                SC_KOM_Server.ResetStep:= TRUE;
                SC_KOM_Server.Step:= 23;
            END_IF

        23:
            SC_KOM_Server.StepName:= '23 - Priradenie QR kodu - odpoved servera';
            SC_KOM_Server.IdleTime.PT:= T#3s;
            SC_KOM_Server.AlarmTime.PT:= T#20s;
            SC_KOM_Server.AlarmTime.IN:= TRUE;

            IF SKTcpClientTrace_1.Status.staReceived AND
                (TRCB_P4_Vytah_ST10.OUTPUTS.TYP_Prikazu = TRCB_P4_Vytah_ST10.INPUTS.TYP_Prikazu) AND
                (TRCB_P4_Vytah_ST10.OUTPUTS.QRkodPowerCP = TRCB_P4_Vytah_ST10.INPUTS.QRkodPowerCP) THEN
                TRCB_P4_Vytah_ST10.STATUS.KomunikaciaUkoncena:= TRUE;
                SC_KOM_Server.ResetStep:= TRUE;
                SC_KOM_Server.Step:= 25;
            ELSIF SC_KOM_Server.AlarmTime.Q THEN
                TRCB_P4_Vytah_ST10.STATUS.KomunikaciaError:= TRUE;
                SC_KOM_Server.ResetStep:= TRUE;
                SC_KOM_Server.Step:= 25;
            END_IF

        25:
            SC_KOM_Server.StepName:= '25 - Vyziadanie stavu paletky - cakam na ukoncenie komunikacie';
            SC_KOM_Server.IdleTime.PT:= T#3s;
            SC_KOM_Server.AlarmTime.PT:= T#10s;

            IF NOT TRCB_P4_Vytah_ST10.CMD.PriradQRkodFiltra_TYP3 THEN
                SC_KOM_Server.ResetStep:= TRUE;
                SC_KOM_Server.Step:= 0;
            END_IF

        30:
            SC_KOM_Server.StepName:= '30 - Vyziadanie serioveho cisla - odoslanie dat na server';
            SC_KOM_Server.IdleTime.PT:= T#3s;
            SC_KOM_Server.AlarmTime.PT:= T#10s;

            TRCB_P4_Vytah_ST10.INPUTS.TYP_Prikazu:= '0';
            TRCB_P4_Vytah_ST10.INPUTS.CisloStanice:= 'ST10';
            TRCB_P4_Vytah_ST10.INPUTS.CisloPaletky;
            TRCB_P4_Vytah_ST10.INPUTS.QRkodPowerCP:= '';
            TRCB_P4_Vytah_ST10.INPUTS.QRkodFiltra:= '';
            TRCB_P4_Vytah_ST10.INPUTS.ID_Operatora:= 'E2';
            TRCB_P4_Vytah_ST10.INPUTS.Report:= '';
            TRCB_P4_Vytah_ST10.INPUTS.StavPaletky:= 'OK';
            SKTcpClientTrace_1.Cmd.Send:= TRUE;

            IF SKTcpClientTrace_1.Cmd.Send AND NOT SKTcpClientTrace_1.Status.staReceived AND NOT SKTcpClientTrace_1.Status.staError THEN
                SC_KOM_Server.ResetStep:= TRUE;
                SC_KOM_Server.Step:= 33;
            END_IF

        33:
            SC_KOM_Server.StepName:= '33 - Vyziadanie serioveho cisla - odpoved servera';
            SC_KOM_Server.IdleTime.PT:= T#3s;
            SC_KOM_Server.AlarmTime.PT:= T#20s;
            SC_KOM_Server.AlarmTime.IN:= TRUE;

            IF SKTcpClientTrace_1.Status.staReceived AND
                (TRCB_P4_Vytah_ST10.OUTPUTS.TYP_Prikazu = TRCB_P4_Vytah_ST10.INPUTS.TYP_Prikazu) THEN
                TRCB_P4_Vytah_ST10.STATUS.KomunikaciaUkoncena:= TRUE;
                SC_KOM_Server.ResetStep:= TRUE;
                SC_KOM_Server.Step:= 35;
            ELSIF SC_KOM_Server.AlarmTime.Q THEN
                TRCB_P4_Vytah_ST10.STATUS.KomunikaciaError:= TRUE;
                SC_KOM_Server.ResetStep:= TRUE;
                SC_KOM_Server.Step:= 35;
            END_IF

        35:
            SC_KOM_Server.StepName:= '35 - Vyziadanie serioveho cisla - cakam na ukoncenie komunikacie';
            SC_KOM_Server.IdleTime.PT:= T#3s;
            SC_KOM_Server.AlarmTime.PT:= T#10s;

            IF NOT TRCB_P4_Vytah_ST10.CMD.VyziadajCisloEtikety_TYP0 THEN
                SC_KOM_Server.ResetStep:= TRUE;
                SC_KOM_Server.Step:= 0;
            END_IF

        40:
            SC_KOM_Server.StepName:= '40 - Odoslanie stavu paletky - odoslanie dat na server';
            SC_KOM_Server.IdleTime.PT:= T#3s;
            SC_KOM_Server.AlarmTime.PT:= T#20s;
            SC_KOM_Server.AlarmTime.IN:= TRUE;

            IF NOT SC_KOM_Server.Switch1 THEN
                brsmemset(ADR(Report),0,SIZEOF(Report));
				brsmemset(ADR(TRCB_P4_Vytah_ST10.INPUTS.Report), 0, SIZEOF(TRCB_P4_Vytah_ST10.INPUTS.Report));

				//Kamera 16//
                Report[0].PoradoveCislo:= '1';
                Report[0].Popis:= 'KAM_16_KontrolaPaletky';
                Report[0].FormatHodnoty:= '2';
                Report[0].Tolerancia_MIN_Hodnota:= '';
                Report[0].Tolerancia_MAX_Hodnota:= '';
                Report[0].Nominal:= 'OK';
                Report[0].Tolerancia_MIN_Jednotky:= '';
                Report[0].Tolerancia_MAX_Jednotky:= '';
                IF Reports.Kamery.P4_CAM16_KontrolaPaletky = 'PASS' THEN
                    Report[0].NameranaHodnota:= 'OK';
                ELSE
                    Report[0].NameranaHodnota:= 'NG';
                END_IF
                Report[0].NameranaHodnota_Jednotky:= '';
                Report[0].VyslednyResult:= Reports.Kamery.P4_CAM16_KontrolaPaletky;
                SKTcpClientNewCsvEntry(Report[0].PoradoveCislo,Report[0].Popis,Report[0].FormatHodnoty,Report[0].Tolerancia_MIN_Hodnota,Report[0].Tolerancia_MAX_Hodnota,Report[0].Nominal,Report[0].Tolerancia_MIN_Jednotky,Report[0].Tolerancia_MAX_Jednotky,Report[0].NameranaHodnota,Report[0].NameranaHodnota_Jednotky,Report[0].VyslednyResult, ADR(TRCB_P4_Vytah_ST10.INPUTS.Report));
                SC_KOM_Server.Switch1:= TRUE;
            END_IF

			TRCB_P4_Vytah_ST10.INPUTS.CisloPaletky:= 'Pal';
			brsstrcat(ADR(TRCB_P4_Vytah_ST10.INPUTS.CisloPaletky), ADR(P4_Vytah.PAR.CisloPaletky_STRING));

            TRCB_P4_Vytah_ST10.INPUTS.TYP_Prikazu:= '2';
            TRCB_P4_Vytah_ST10.INPUTS.CisloStanice:= 'ST10';
            TRCB_P4_Vytah_ST10.INPUTS.QRkodPowerCP:= Paletka[a].PAR.QRkodPowerCP;
            TRCB_P4_Vytah_ST10.INPUTS.QRkodFiltra:= '';
            TRCB_P4_Vytah_ST10.INPUTS.ID_Operatora:= Paletka[a].PAR.ID_Operatora;
            TRCB_P4_Vytah_ST10.INPUTS.Report:= '';
            TRCB_P4_Vytah_ST10.INPUTS.StavPaletky:= Paletka[a].PAR.StavPowerCP;

			IF SKTcpClientTrace_1.Status.staReadyToSend AND NOT SKTcpClientTrace_1.Cmd.Close THEN
				TRCB_P4_Vytah_ST10.OUTPUTS.TYP_Prikazu:= '';
				SKTcpClientTrace_1.Cmd.Send:= TRUE;
				SC_KOM_Server.ResetStep:= TRUE;
				SC_KOM_Server.Step:= 43;
			END_IF

        43:
            SC_KOM_Server.StepName:= '43 - Odoslanie stavu paletky - odpoved servera';
			SC_KOM_Server.IdleTime.PT:= T#3s;
            SC_KOM_Server.AlarmTime.PT:= T#7s;
            SC_KOM_Server.AlarmTime.IN:= TRUE;

            IF SKTcpClientTrace_1.Status.staReceived AND
                (TRCB_P4_Vytah_ST10.OUTPUTS.TYP_Prikazu = TRCB_P4_Vytah_ST10.INPUTS.TYP_Prikazu) AND
                (TRCB_P4_Vytah_ST10.OUTPUTS.QRkodPowerCP = TRCB_P4_Vytah_ST10.INPUTS.QRkodPowerCP) THEN
                TRCB_P4_Vytah_ST10.STATUS.KomunikaciaUkoncena:= TRUE;
                SC_KOM_Server.ResetStep:= TRUE;
                SC_KOM_Server.Step:= 45;
            ELSIF SC_KOM_Server.AlarmTime.Q AND NOT SKTcpClientTrace_1.Status.staSending THEN
                PocetDopytovNaServer:= PocetDopytovNaServer + 1;
				SKTcpClientTrace_1.Cmd.Send:= FALSE;
				SKTcpClientTrace_1.Cmd.Close:= TRUE;
				SC_KOM_Server.ResetStep:= TRUE;
                SC_KOM_Server.Step:= 44;
            END_IF

        44:
            SC_KOM_Server.StepName:= '44 - Odoslanie stavu paletky - cakam na opatovny dopyt na server';
            SC_KOM_Server.IdleTime.PT:= T#1s;
            SC_KOM_Server.AlarmTime.PT:= T#10s;
            SC_KOM_Server.IdleTime.IN:= TRUE;
            SKTcpClientTrace_1.Cmd.Send:= FALSE;

            IF PocetDopytovNaServer < 3 THEN
                IF SC_KOM_Server.IdleTime.Q THEN
                    SC_KOM_Server.ResetStep:= TRUE;
                    SC_KOM_Server.Step:= 40;
                END_IF
            ELSE
                TRCB_P4_Vytah_ST10.STATUS.KomunikaciaError:= TRUE;
                SC_KOM_Server.ResetStep:= TRUE;
                SC_KOM_Server.Step:= 45;
            END_IF

        45:
            SC_KOM_Server.StepName:= '45 - Vyziadanie serioveho cisla - cakam na ukoncenie komunikacie';
            SC_KOM_Server.IdleTime.PT:= T#3s;
            SC_KOM_Server.AlarmTime.PT:= T#10s;

            IF NOT TRCB_P4_Vytah_ST10.CMD.OdosliStavPaletky_TYP2 THEN
                SC_KOM_Server.ResetStep:= TRUE;
                SC_KOM_Server.Step:= 0;
            END_IF

		50:
			SC_KOM_Server.StepName:= '50 - Vyziadanie stavu Panatrace - odoslanie dat na server';
			SC_KOM_Server.IdleTime.PT:= T#3s;
			SC_KOM_Server.AlarmTime.PT:= T#10s;
			SC_KOM_Server.AlarmTime.IN:= TRUE;

			TRCB_P4_Vytah_ST10.INPUTS.TYP_Prikazu:= '4';
			TRCB_P4_Vytah_ST10.INPUTS.CisloStanice:= 'ST10';
			TRCB_P4_Vytah_ST10.INPUTS.CisloPaletky:= '';
			TRCB_P4_Vytah_ST10.INPUTS.QRkodPowerCP:= '';
			TRCB_P4_Vytah_ST10.INPUTS.QRkodFiltra:= '';
			TRCB_P4_Vytah_ST10.INPUTS.ID_Operatora:= '';
			TRCB_P4_Vytah_ST10.INPUTS.Report:= '';
			TRCB_P4_Vytah_ST10.INPUTS.StavPaletky:= '';

			IF SKTcpClientTrace_1.Status.staReadyToSend AND NOT SKTcpClientTrace_1.Cmd.Close THEN
				TRCB_P4_Vytah_ST10.OUTPUTS.TYP_Prikazu:= '';
				SKTcpClientTrace_1.Cmd.Send:= TRUE;
				SC_KOM_Server.ResetStep:= TRUE;
				SC_KOM_Server.Step:= 53;
			END_IF

		53:
			SC_KOM_Server.StepName:= '53 - Vyziadanie stavu paletky - odpoved servera';
			SC_KOM_Server.IdleTime.PT:= T#30s;
			SC_KOM_Server.AlarmTime.PT:= T#7s;
			SC_KOM_Server.AlarmTime.IN:= TRUE;

			IF SKTcpClientTrace_1.Status.staReceived AND TRCB_P4_Vytah_ST10.OUTPUTS.TYP_Prikazu = TRCB_P4_Vytah_ST10.INPUTS.TYP_Prikazu THEN
				TRCB_P4_Vytah_ST10.STATUS.KomunikaciaUkoncena:= TRUE;
				SC_KOM_Server.ResetStep:= TRUE;
				SC_KOM_Server.Step:= 55;
			ELSIF SC_KOM_Server.AlarmTime.Q AND NOT SKTcpClientTrace_1.Status.staSending THEN
				PocetDopytovNaServer:= PocetDopytovNaServer + 1;
				SKTcpClientTrace_1.Cmd.Send:= FALSE;
				SKTcpClientTrace_1.Cmd.Close:= TRUE;
				SC_KOM_Server.ResetStep:= TRUE;
				SC_KOM_Server.Step:= 54;
			END_IF

		54:
			SC_KOM_Server.StepName:= '54 - Vyziadanie stavu paletky - cakam na opatovny dopyt na server';
			SC_KOM_Server.IdleTime.PT:= T#1s;
			SC_KOM_Server.AlarmTime.PT:= T#10s;
			SC_KOM_Server.IdleTime.IN:= TRUE;

			IF PocetDopytovNaServer < 3 THEN
				IF SC_KOM_Server.IdleTime.Q THEN
					SC_KOM_Server.ResetStep:= TRUE;
					SC_KOM_Server.Step:= 50;
				END_IF
			ELSE
				TRCB_P4_Vytah_ST10.STATUS.KomunikaciaError:= TRUE;
				SC_KOM_Server.ResetStep:= TRUE;
				SC_KOM_Server.Step:= 55;
			END_IF

		55:
			SC_KOM_Server.StepName:= '55 - Vyziadanie stavu paletky - cakam na ukoncenie komunikacie';
			SC_KOM_Server.IdleTime.PT:= T#3s;
			SC_KOM_Server.AlarmTime.PT:= T#10s;

			IF NOT TRCB_P4_Vytah_ST10.CMD.VyziadajStavPanatrace_TYP4 THEN
				SC_KOM_Server.ResetStep:= TRUE;
				SC_KOM_Server.Step:= 0;
			END_IF

    END_CASE

END_PROGRAM

PROGRAM _EXIT
	(* Insert code here *)

END_PROGRAM
```

#### Types.typ - Local data types
```iecst
TYPE
	Report_typ : 	STRUCT
		PoradoveCislo : STRING[2]; (*IDstep - Poradové čislo reportu*)
		Popis : STRING[100]; (*Description - Popis*)
		FormatHodnoty : STRING[2]; (*TypValue - Format zaslané hodnoty  1- Číslo, 2 - Znak*)
		Tolerancia_MIN_Hodnota : STRING[10]; (*MinTol - Minimálna tolerancia meranej veličiny*)
		Tolerancia_MAX_Hodnota : STRING[10]; (*MaxTol - Maximálna tolerancia meranej veličiny*)
		Nominal : STRING[10]; (*Nom - Ak jezvolený formát string tak tu zadáme OK inak je prazdna*)
		Tolerancia_MIN_Jednotky : STRING[10]; (*MinEle - Jednotky minimálnej tolerancie veličiny*)
		Tolerancia_MAX_Jednotky : STRING[10]; (*MaxEle - Jednotky maximálnej tolerancie veličiny*)
		NameranaHodnota : STRING[10]; (*Value - Namerana hodnota veličiny, ak su kamery tak bude hodnota OK alebo NG*)
		NameranaHodnota_Jednotky : STRING[10]; (*ValEle - Jednotky nameranej veličiny*)
		VyslednyResult : STRING[5]; (*Result - Výsledný result  PASS, FAIL, SKIP*)
	END_STRUCT;
END_TYPE
```

#### Variables.var - Local variables
```iecst
VAR
	SC_KOM_Server : SequenceControlTyp;
	SKTcpClientTrace_1 : SKTcpClientTrace;
	a : USINT;
	Report : ARRAY[0..50] OF Report_typ;
	PocetDopytovNaServer : USINT;
END_VAR
```

### Program Logical/Blikace/Blikanie100ms (IEC)

#### Blikanie100ms.st - Init, cyclic, exit code
```iecst
PROGRAM _INIT
	(* Insert code here *)

END_PROGRAM

PROGRAM _CYCLIC

	IF NOT Blikac100ms THEN
		Blikac100ms:= TRUE;
	ELSE
		Blikac100ms:= FALSE;
	END_IF

END_PROGRAM

PROGRAM _EXIT
	(* Insert code here *)

END_PROGRAM
```

### Program Logical/Blikace/Blikanie200ms (IEC)

#### Blikanie200ms.st - Init, cyclic, exit code
```iecst
PROGRAM _INIT
	(* Insert code here *)

END_PROGRAM

PROGRAM _CYCLIC

	IF NOT Blikac200ms THEN
		Blikac200ms:= TRUE;
	ELSE
		Blikac200ms:= FALSE;
	END_IF

END_PROGRAM

PROGRAM _EXIT
	(* Insert code here *)

END_PROGRAM
```

### Program Logical/Blikace/Blikanie500ms (IEC)

#### Blikanie500ms.st - Init, cyclic, exit code
```iecst
PROGRAM _INIT
	(* Insert code here *)

END_PROGRAM

PROGRAM _CYCLIC
	IF NOT Blikac500ms THEN
		Blikac500ms:= TRUE;
	ELSE
		Blikac500ms:= FALSE;
	END_IF

END_PROGRAM

PROGRAM _EXIT
	(* Insert code here *)

END_PROGRAM
```

### Program Logical/Blikace/Blikanie1s (IEC)

#### Blikanie1s.st - Init, cyclic, exit code
```iecst
PROGRAM _INIT
	(* Insert code here *)

END_PROGRAM

PROGRAM _CYCLIC
	IF NOT Blikac1s THEN
		Blikac1s:= TRUE;
	ELSE
		Blikac1s:= FALSE;
	END_IF

END_PROGRAM

PROGRAM _EXIT
	(* Insert code here *)

END_PROGRAM
```

### UsersGlobal.typ - Global data types
```iecst
TYPE
	UsersVizu_typ : 	STRUCT
		TypPrihlasenia : USINT;
		ZoznamUzivatelov : ARRAY[0..100]OF STRING[100];
		Edit_MenoUzivatela : STRING[80]; (*Meno zadavané pri uložení uživatela*)
		Edit_HesloUzivatela : STRING[80]; (*Heslo zadané pri uložení uživatela*)
		Edit_CisloKarty : STRING[80]; (*Cislo karty nacitane pri uložení uživatela*)
		Edit_UrovenUzivatela : STRING[80];
		CisloPrihlasenejKarty_Panel1 : STRING[80]; (*Cislo karty nacitane pri uložení uživatela*)
		CisloPrihlasenejKarty_Panel2 : STRING[80]; (*Cislo karty nacitane pri uložení uživatela*)
		CisloPrihlasenejKarty_Panel3 : STRING[80]; (*Cislo karty nacitane pri uložení uživatela*)
		ZadaneMenoUzivatela : STRING[80]; (*Meno zadané cez prihlasovacie okno*)
		ZadaneHesloUzivatela : STRING[80]; (*Heslo zadané cez prihlasovacie okno*)
		ZadaneCisloKarty_Panel1 : STRING[80]; (*Cislo karty načítané pri prihlásení*)
		ZadaneCisloKarty_Panel2 : STRING[80]; (*Cislo karty načítané pri prihlásení*)
		ZadaneCisloKarty_Panel3 : STRING[80]; (*Cislo karty načítané pri prihlásení*)
		MenoPrihlasenehoUzivatela_Panel1 : STRING[80]; (*Zobrazuje sa vo vizualizácii*)
		MenoPrihlasenehoUzivatela_Panel2 : STRING[80]; (*Zobrazuje sa vo vizualizácii*)
		MenoPrihlasenehoUzivatela_Panel3 : STRING[80]; (*Zobrazuje sa vo vizualizácii*)
		UlozUzivatela : BOOL;
		PrihlasUzivatela : BOOL;
		VymazUzivatela : BOOL;
		OdhlasUzivatela_Panel1 : BOOL;
		OdhlasUzivatela_Panel2 : BOOL;
		OdhlasUzivatela_Panel3 : BOOL;
		NacitajUzivatela : BOOL;
		LB_Index : UINT;
		LB_IndexSTRING : STRING[80];
		KartaPrilozena_Panel1 : BOOL;
		KartaPrilozena_Panel2 : BOOL;
		KartaPrilozena_Panel3 : BOOL;
		EditaciaMena_ENABLE : BOOL;
		EditaciaHesla_ENABLE : BOOL;
		EditaciaKarty_ENABLE : BOOL;
		TL_UlozUzivatela_ENABLE : BOOL;
		TL_VymazUzivatela_ENABLE : BOOL;
		TlacitkoPrihlasenie_ENABLE : BOOL;
		Stav_ExistujuciUzivatel : BOOL;
		Stav_ChybajuceDataUzivatela : BOOL;
		StavyUsers_Index : USINT;
	END_STRUCT;
	ParametreUzivatelovTyp : 	STRUCT
		Meno : STRING[80];
		Heslo : STRING[80];
		CisloKarty : STRING[80];
		UrovenUzivatela : UINT;
	END_STRUCT;
END_TYPE
```

### UsersGlobal.var - Global variables
```iecst
VAR
	UsersVizu : UsersVizu_typ;
	MpRecipeXml_1 : MpRecipeXml := (0);
	MpRecipeRegPar_1 : MpRecipeRegPar := (0);
	Uzivatel : ARRAY[0..100] OF ParametreUzivatelovTyp;
	PrecitaneData_Panel1 : ARRAY[0..19] OF UDINT;
	PrecitaneData_Panel2 : ARRAY[0..19] OF UDINT;
	PrecitaneData_Panel3 : ARRAY[0..19] OF UDINT;
	PrecitaneData_Panel4 : ARRAY[0..19] OF UDINT;
	CisloPrihlasenejKarty_Panel1 : STRING[80];
	P1_UzivatelPrihlaseny : BOOL;
	P1_UrovenPrihlasenehoUzivatela : UINT; (*10 - operator, 20 - technik, 100 - administrátor*)
	P2_UzivatelPrihlaseny : BOOL;
	P2_UrovenPrihlasenehoUzivatela : UINT; (*10 - operator, 20 - technik, 100 - administrátor*)
	P34_UzivatelPrihlaseny : BOOL;
	P34_UrovenPrihlasenehoUzivatela : UINT; (*10 - operator, 20 - technik, 100 - administrátor*)
	Citacka1_AKTIVNA : BOOL;
	Citacka2_AKTIVNA : BOOL;
	Citacka3_AKTIVNA : BOOL;
END_VAR
```

### Program Logical/Uzivatelia/RFID_Prg (IEC)

#### RFID_Prg.st - Implementation code
```iecst
(********************************************************************
 * COPYRIGHT -- Bernecker + Rainer
 ********************************************************************
 * Program: RFID_Prg
 * File: RFID_Prg.st
 * Author: borsm
 * Created: December 23, 2015
 ********************************************************************
 * Implementation of program RFID_Prg
 ********************************************************************)

PROGRAM _INIT

    doinit:=1;

END_PROGRAM

PROGRAM _CYCLIC

	//Reset čitačiek RFID//
    IF NOT CasResetovaniaCitaciekRFID.Q THEN
        CasResetovaniaCitaciekRFID.IN:= TRUE;
    ELSIF CasResetovaniaCitaciekRFID.Q THEN
        doinit:= TRUE;
        CasResetovaniaCitaciekRFID.IN:= FALSE;
    END_IF

    CasResetovaniaCitaciekRFID.PT:= T#5m;
    CasResetovaniaCitaciekRFID();

(* find the Transponder, and give the Device ID back, this FuB works only for USB interface Transponder,

IF you use a serial interface transponder, please give the adress OF Interface ID directly TO the ident OF all FuBs *)

//Hladanie RFID čitačky//
    IF doinit THEN
        InitDone:= FALSE;
        doRead:= FALSE;
        TP_Init_0.Enable := TRUE;
        IF TP_Init_0.Done THEN
            PoruchaVyhladaniaCitaciek:= FALSE;
            DeviceID1 := TP_Init_0.Ident[2]; //Panel č.1
            DeviceID2 := TP_Init_0.Ident[1]; //Panel č.2
            DeviceID3 := TP_Init_0.Ident[0]; //Panel č.3
            TP_Init_0.Enable := FALSE;
            poc := poc + 1;
            IF poc	>= 3 THEN
                InitDone:= TRUE;
                doRead := TRUE;
                doinit:= FALSE;
                poc := 0;
            END_IF
        ELSIF TP_Init_0.Error THEN
            PoruchaVyhladaniaCitaciek:= TRUE;
            TP_Init_0.Enable := FALSE;
            doRead:= FALSE;
            doinit := FALSE;
        END_IF
    END_IF

    (* Čítanie z čítačky *)

    IF doRead AND InitDone AND NOT InitError THEN

        //Panel 1//
        TP_Read_1.Ident := DeviceID1;
        TP_Read_1.Enable := TRUE;
        IF TP_Read_1.Done THEN
            strcpy(ADR(READDATA_Citacka1),TP_Read_1.Data);
            TP_Read_1.Enable := FALSE;
        ELSIF TP_Read_1.Error THEN
            memset(ADR(READDATA_Citacka1),0,SIZEOF(READDATA_Citacka1));
            TP_Read_1.Enable := FALSE;
        END_IF

        //Panel 2//
        TP_Read_2.Ident := DeviceID2;
        TP_Read_2.Enable := TRUE;
        IF TP_Read_2.Done THEN
            strcpy(ADR(READDATA_Citacka2),TP_Read_2.Data);
            TP_Read_2.Enable := FALSE;
        ELSIF TP_Read_2.Error THEN
            memset(ADR(READDATA_Citacka2),0,SIZEOF(READDATA_Citacka2));
            TP_Read_2.Enable := FALSE;
        END_IF

        //Panel 3//
        TP_Read_3.Ident := DeviceID3;
        TP_Read_3.Enable := TRUE;
        IF TP_Read_3.Done THEN
           strcpy(ADR(READDATA_Citacka3),TP_Read_3.Data);
           TP_Read_3.Enable := FALSE;
        ELSIF TP_Read_3.Error THEN
           memset(ADR(READDATA_Citacka3),0,SIZEOF(READDATA_Citacka3));
           TP_Read_3.Enable := FALSE;
        END_IF

    ELSE
        TP_Read_1.Enable := FALSE;
        TP_Read_2.Enable := FALSE;
        TP_Read_3.Enable := FALSE;
        memset(ADR(READDATA_Citacka1),0,SIZEOF(READDATA_Citacka1));
        memset(ADR(READDATA_Citacka2),0,SIZEOF(READDATA_Citacka2));
        memset(ADR(READDATA_Citacka3),0,SIZEOF(READDATA_Citacka3));
    END_IF

    (* call FuBs *)
    TP_Init_0();
    TP_Read_1();
    TP_Read_2();
    TP_Read_3();

    //Zistenie či je priložená karta na čitačke 1//
    IF READDATA_Citacka1[2] = 0
        AND READDATA_Citacka1[3] = 0
        AND READDATA_Citacka1[4] = 0
        AND READDATA_Citacka1[5] = 0
        AND READDATA_Citacka1[6] = 0
        AND READDATA_Citacka1[7] = 0
        AND READDATA_Citacka1[8] = 0
        AND READDATA_Citacka1[9] = 0 THEN
        Citacka1_AKTIVNA:= FALSE;
    ELSE
        Citacka1_AKTIVNA:= TRUE;
    END_IF

    //Zistenie či je priložená karta na čitačke 2//
    IF READDATA_Citacka2[2] = 0
        AND READDATA_Citacka2[3] = 0
        AND READDATA_Citacka2[4] = 0
        AND READDATA_Citacka2[5] = 0
        AND READDATA_Citacka2[6] = 0
        AND READDATA_Citacka2[7] = 0
        AND READDATA_Citacka2[8] = 0
        AND READDATA_Citacka2[9] = 0 THEN
        Citacka2_AKTIVNA:= FALSE;
    ELSE
        Citacka2_AKTIVNA:= TRUE;
    END_IF

    //Zistenie či je priložená karta na čitačke 3//
    IF READDATA_Citacka3[2] = 0
        AND READDATA_Citacka3[3] = 0
        AND READDATA_Citacka3[4] = 0
        AND READDATA_Citacka3[5] = 0
        AND READDATA_Citacka3[6] = 0
        AND READDATA_Citacka3[7] = 0
        AND READDATA_Citacka3[8] = 0
        AND READDATA_Citacka3[9] = 0 THEN
        Citacka3_AKTIVNA:= FALSE;
    ELSE
        Citacka3_AKTIVNA:= TRUE;
    END_IF

    //Načítané kódy čitačiek//
    //Panel 1//
    IF P1_Vizu.TL_PrihlasovOperatora_AKTIVNE THEN  //Panel 1//
        IF Citacka1_AKTIVNA THEN
            PrecitaneData_Panel1[0]:= READDATA_Citacka1[3];
            PrecitaneData_Panel1[1]:= READDATA_Citacka1[2];
            PrecitaneData_Panel1[2]:= READDATA_Citacka1[5];
            PrecitaneData_Panel1[3]:= READDATA_Citacka1[4];
            PrecitaneData_Panel1[4]:= READDATA_Citacka1[7];
            PrecitaneData_Panel1[5]:= READDATA_Citacka1[6];
            PrecitaneData_Panel1[6]:= READDATA_Citacka1[9];
            PrecitaneData_Panel1[7]:= READDATA_Citacka1[8];
        ELSIF Citacka2_AKTIVNA THEN
            PrecitaneData_Panel1[0]:= READDATA_Citacka2[3];
            PrecitaneData_Panel1[1]:= READDATA_Citacka2[2];
            PrecitaneData_Panel1[2]:= READDATA_Citacka2[5];
            PrecitaneData_Panel1[3]:= READDATA_Citacka2[4];
            PrecitaneData_Panel1[4]:= READDATA_Citacka2[7];
            PrecitaneData_Panel1[5]:= READDATA_Citacka2[6];
            PrecitaneData_Panel1[6]:= READDATA_Citacka2[9];
            PrecitaneData_Panel1[7]:= READDATA_Citacka2[8];
        ELSIF Citacka3_AKTIVNA THEN
            PrecitaneData_Panel1[0]:= READDATA_Citacka3[3];
            PrecitaneData_Panel1[1]:= READDATA_Citacka3[2];
            PrecitaneData_Panel1[2]:= READDATA_Citacka3[5];
            PrecitaneData_Panel1[3]:= READDATA_Citacka3[4];
            PrecitaneData_Panel1[4]:= READDATA_Citacka3[7];
            PrecitaneData_Panel1[5]:= READDATA_Citacka3[6];
            PrecitaneData_Panel1[6]:= READDATA_Citacka3[9];
            PrecitaneData_Panel1[7]:= READDATA_Citacka3[8];
        END_IF
    ELSIF P2_Vizu.TL_PrihlasovOperatora_AKTIVNE THEN  //Panel 2//
        IF Citacka1_AKTIVNA THEN
            PrecitaneData_Panel2[0]:= READDATA_Citacka1[3];
            PrecitaneData_Panel2[1]:= READDATA_Citacka1[2];
            PrecitaneData_Panel2[2]:= READDATA_Citacka1[5];
            PrecitaneData_Panel2[3]:= READDATA_Citacka1[4];
            PrecitaneData_Panel2[4]:= READDATA_Citacka1[7];
            PrecitaneData_Panel2[5]:= READDATA_Citacka1[6];
            PrecitaneData_Panel2[6]:= READDATA_Citacka1[9];
            PrecitaneData_Panel2[7]:= READDATA_Citacka1[8];
        ELSIF Citacka2_AKTIVNA THEN
            PrecitaneData_Panel2[0]:= READDATA_Citacka2[3];
            PrecitaneData_Panel2[1]:= READDATA_Citacka2[2];
            PrecitaneData_Panel2[2]:= READDATA_Citacka2[5];
            PrecitaneData_Panel2[3]:= READDATA_Citacka2[4];
            PrecitaneData_Panel2[4]:= READDATA_Citacka2[7];
            PrecitaneData_Panel2[5]:= READDATA_Citacka2[6];
            PrecitaneData_Panel2[6]:= READDATA_Citacka2[9];
            PrecitaneData_Panel2[7]:= READDATA_Citacka2[8];
        ELSIF Citacka3_AKTIVNA THEN
            PrecitaneData_Panel2[0]:= READDATA_Citacka3[3];
            PrecitaneData_Panel2[1]:= READDATA_Citacka3[2];
            PrecitaneData_Panel2[2]:= READDATA_Citacka3[5];
            PrecitaneData_Panel2[3]:= READDATA_Citacka3[4];
            PrecitaneData_Panel2[4]:= READDATA_Citacka3[7];
            PrecitaneData_Panel2[5]:= READDATA_Citacka3[6];
            PrecitaneData_Panel2[6]:= READDATA_Citacka3[9];
            PrecitaneData_Panel2[7]:= READDATA_Citacka3[8];
        END_IF
    ELSIF P34_Vizu.TL_PrihlasovOperatora_AKTIVNE THEN  //Panel 3//
        IF Citacka1_AKTIVNA THEN
            PrecitaneData_Panel3[0]:= READDATA_Citacka1[3];
            PrecitaneData_Panel3[1]:= READDATA_Citacka1[2];
            PrecitaneData_Panel3[2]:= READDATA_Citacka1[5];
            PrecitaneData_Panel3[3]:= READDATA_Citacka1[4];
            PrecitaneData_Panel3[4]:= READDATA_Citacka1[7];
            PrecitaneData_Panel3[5]:= READDATA_Citacka1[6];
            PrecitaneData_Panel3[6]:= READDATA_Citacka1[9];
            PrecitaneData_Panel3[7]:= READDATA_Citacka1[8];
        ELSIF Citacka2_AKTIVNA THEN
            PrecitaneData_Panel3[0]:= READDATA_Citacka2[3];
            PrecitaneData_Panel3[1]:= READDATA_Citacka2[2];
            PrecitaneData_Panel3[2]:= READDATA_Citacka2[5];
            PrecitaneData_Panel3[3]:= READDATA_Citacka2[4];
            PrecitaneData_Panel3[4]:= READDATA_Citacka2[7];
            PrecitaneData_Panel3[5]:= READDATA_Citacka2[6];
            PrecitaneData_Panel3[6]:= READDATA_Citacka2[9];
            PrecitaneData_Panel3[7]:= READDATA_Citacka2[8];
        ELSIF Citacka3_AKTIVNA THEN
            PrecitaneData_Panel3[0]:= READDATA_Citacka3[3];
            PrecitaneData_Panel3[1]:= READDATA_Citacka3[2];
            PrecitaneData_Panel3[2]:= READDATA_Citacka3[5];
            PrecitaneData_Panel3[3]:= READDATA_Citacka3[4];
            PrecitaneData_Panel3[4]:= READDATA_Citacka3[7];
            PrecitaneData_Panel3[5]:= READDATA_Citacka3[6];
            PrecitaneData_Panel3[6]:= READDATA_Citacka3[9];
            PrecitaneData_Panel3[7]:= READDATA_Citacka3[8];
        END_IF
    ELSE
        PrecitaneData_Panel1[0]:= 0;
        PrecitaneData_Panel1[1]:= 0;
        PrecitaneData_Panel1[2]:= 0;
        PrecitaneData_Panel1[3]:= 0;
        PrecitaneData_Panel1[4]:= 0;
        PrecitaneData_Panel1[5]:= 0;
        PrecitaneData_Panel1[6]:= 0;
        PrecitaneData_Panel1[7]:= 0;

        PrecitaneData_Panel2[0]:= 0;
        PrecitaneData_Panel2[1]:= 0;
        PrecitaneData_Panel2[2]:= 0;
        PrecitaneData_Panel2[3]:= 0;
        PrecitaneData_Panel2[4]:= 0;
        PrecitaneData_Panel2[5]:= 0;
        PrecitaneData_Panel2[6]:= 0;
        PrecitaneData_Panel2[7]:= 0;

        PrecitaneData_Panel3[0]:= 0;
        PrecitaneData_Panel3[1]:= 0;
        PrecitaneData_Panel3[2]:= 0;
        PrecitaneData_Panel3[3]:= 0;
        PrecitaneData_Panel3[4]:= 0;
        PrecitaneData_Panel3[5]:= 0;
        PrecitaneData_Panel3[6]:= 0;
        PrecitaneData_Panel3[7]:= 0;
    END_IF

END_PROGRAM
```

#### RFID_Prg.var - Local variables
```iecst
(********************************************************************
 * COPYRIGHT -- Bernecker + Rainer
 ********************************************************************
 * Program: RFID_Prg
 * File: RFID_Prg.var
 * Author: borsm
 * Created: December 23, 2015
 ********************************************************************
 * Local variables of program RFID_Prg
 ********************************************************************)
VAR
	TP_Read_4 : TP_Read;
	TP_Read_1 : TP_Read;
	TP_Read_2 : TP_Read;
	TP_Read_3 : TP_Read;
	DeviceID1 : UDINT;
	DeviceID2 : UDINT;
	DeviceID3 : UDINT;
	DeviceID4 : UDINT;
	READDATA_Citacka1 : ARRAY[0..19] OF USINT;
	READDATA_Citacka2 : ARRAY[0..19] OF USINT;
	READDATA_Citacka3 : ARRAY[0..19] OF USINT;
	READDATA_Citacka4 : ARRAY[0..19] OF USINT;
	TP_Write_0 : TP_Write;
	WRITEDATA : STRING[8];
	ReadDone_Panel1 : BOOL;
	ReadDone_Panel2 : BOOL;
	ReadDone_Panel3 : BOOL;
	ReadError_Panel1 : BOOL;
	ReadError_Panel2 : BOOL;
	ReadError_Panel3 : BOOL;
	ReadErrorID_Panel1 : UDINT;
	ReadErrorID_Panel2 : UDINT;
	ReadErrorID_Panel3 : UDINT;
	doRead : BOOL;
	doWrite : BOOL;
	WriteDone : BOOL;
	WriteError : BOOL;
	WriteErrorID : UDINT;
	TP_Init_0 : TP_Init;
	TP_OnOff_0 : TP_OnOff;
	TP_Crc_0 : TP_Crc;
	TP_Lock_0 : TP_Lock;
	TP_Info_0 : TP_Info;
	TP_PWProtect_0 : TP_PWProtect;
	TP_Unlock_0 : TP_Unlock;
	doPassword : BOOL;
	PasswordErrorID : UDINT;
	PasswordError : BOOL;
	PasswordDone : BOOL;
	passwordin : STRING[8];
	doUnlock : BOOL;
	UnlockErrorID : UDINT;
	UnlockError : BOOL;
	UnlockDone : BOOL;
	password : STRING[8];
	doLock : BOOL;
	LockErrorID : UDINT;
	LockError : BOOL;
	LockDone : BOOL;
	doCrc : BOOL;
	CrcErrorID : UDINT;
	CrcError : BOOL;
	CrcDone : BOOL;
	doInfo : BOOL;
	InfoErrorID : UDINT;
	InfoError : BOOL;
	InfoDone : BOOL;
	sl : ARRAY[0..1] OF USINT;
	KEYTYPE : ARRAY[0..3] OF USINT;
	Type : ARRAY[0..30] OF USINT;
	ID : ARRAY[0..9] OF USINT;
	doOnOff : BOOL;
	OnOffDone : BOOL;
	OnOffErrorID : UDINT;
	OnOffError : BOOL;
	InitDone : BOOL;
	InitErrorID : UDINT;
	InitError : BOOL;
	poc : USINT;
	step : INT;
	doinit : BOOL;
	CasResetovaniaCitaciekRFID : TON;
	PoruchaVyhladaniaCitaciek : BOOL;
	TEST : BOOL;
	a : USINT;
	b : USINT;
	c : USINT;
END_VAR
```

### Program Logical/Uzivatelia/Users_Main (IEC)

#### Main.st - Init, cyclic, exit code
```iecst
PROGRAM _INIT
	MpRecipeXml_1.Load:= TRUE;

END_PROGRAM

PROGRAM _CYCLIC

	//Volanie funkcie SequenceControl//
	SequenceControl(SC:= SC_Uzivatelia);

	//Načítanie receptur z pamäte//
	IF MpRecipeXml_1.Load AND (MpRecipeXml_1.CommandDone OR MpRecipeXml_1.Error) THEN
		MpRecipeXml_1.Load:= FALSE;
	END_IF

	//Konfigurácia receptur//
	MpRecipeXml_1.MpLink:= ADR(gUserXml);  //takto sa menuje mapp komponenta v configurating view//
	MpRecipeXml_1.Enable:= TRUE;
	MpRecipeXml_1.Category:= ADR('UZIVATELIA');
	MpRecipeXml_1.Category:= ADR(strCategory);
	MpRecipeXml_1.DeviceName:= ADR('HDD_Users');  //Názov media, kde sa budú receptury ukladat//
	MpRecipeXml_1.FileName:= ADR('UlozeniUzivatelia'); //Názov súboru do ktorého sa receptúry uložia//
	MpRecipeXml_1();

	MpRecipeRegPar_1.MpLink:= ADR(gUserXml);
	MpRecipeRegPar_1.Enable:= TRUE;
	MpRecipeRegPar_1.Category:= ADR('UZIVATELIA');
	MpRecipeRegPar_1.PVName:= ADR('Uzivatel'); //Názov premenné, kde je vytvorená štruktura dat pre receptury//
	MpRecipeRegPar_1();

    //Zamknutie tlačítka Uloženie uživatelov//
    IF UsersVizu.Edit_MenoUzivatela = '' THEN
        UsersVizu.TL_UlozUzivatela_ENABLE:= FALSE;
    ELSIF UsersVizu.Edit_CisloKarty = '' THEN
        UsersVizu.TL_UlozUzivatela_ENABLE:= FALSE;
    ELSE
        UsersVizu.TL_UlozUzivatela_ENABLE:= TRUE;
   END_IF

    //Zobrazenie zoznamu uživatelov//

    FOR a:= 0 TO 100 BY 1 DO
        ListBoxPole_Sprava[a]:= '{"value":"';
        ListBox_Value[a]:= UINT_TO_STRING(a);
        brsstrcat(ADR(ListBoxPole_Sprava[a]), ADR(ListBox_Value[a]));
        brsstrcat(ADR(ListBoxPole_Sprava[a]), ADR('","text":"'));
        brsstrcat(ADR(ListBoxPole_Sprava[a]), ADR(Uzivatel[a].Meno));
        brsstrcat(ADR(ListBoxPole_Sprava[a]), ADR('"}'));
        IF Uzivatel[a].Meno = '' THEN
            UsersVizu.ZoznamUzivatelov[a]:= '';
        ELSE
            UsersVizu.ZoznamUzivatelov[a]:= ListBoxPole_Sprava[a];
        END_IF
    END_FOR

    //Vyčítanie aktuálneho indexu text listu (hodnota string) a prevod do premennej UINT//
    e:= STRING_TO_UINT(UsersVizu.LB_IndexSTRING);

    //Načítanie čísla karty//
    IF P1_Vizu.TL_PrihlasovOperatora_AKTIVNE AND (Citacka1_AKTIVNA OR Citacka2_AKTIVNA OR Citacka3_AKTIVNA) THEN
        UsersVizu.Edit_CisloKarty:= CisloPrihlasenejKarty_Panel1;
    END_IF

    IF NOT P1_Vizu.TL_PrihlasovOperatora_AKTIVNE THEN
        UsersVizu.Edit_CisloKarty:= '';
    END_IF

    //***************************************Editácia databáze uzivatelov*********************************//
    CASE SC_Uzivatelia.Step OF

        0://Vynulovanie uživatela//
            SC_Uzivatelia.StepName:= '0 - Nulovanie';
            UsersVizu.UlozUzivatela:= FALSE;
            UsersVizu.VymazUzivatela:= FALSE;
            UsersVizu.NacitajUzivatela:= FALSE;

            MpRecipeXml_1.Save:= FALSE;
            i:= 0;
            c:= 0;
            d:= 0;
            IndexPrazdPole:= 0;
            SC_Uzivatelia.ResetStep:= TRUE;
            SC_Uzivatelia.Step:= 1;

        1://Rozhodnutie o činnosti//
            SC_Uzivatelia.StepName:= '1 - Rozhodnutie o cinnosti';
            IF UsersVizu.UlozUzivatela THEN
                SC_Uzivatelia.Step:= 10;
            ELSIF UsersVizu.NacitajUzivatela THEN
                SC_Uzivatelia.Step:= 20;
            ELSIF UsersVizu.VymazUzivatela THEN
                SC_Uzivatelia.Step:= 30;
            END_IF

        10://Kontrola zadaných udajov uzivatela//
            SC_Uzivatelia.StepName:= '10 - Kontrola zadanych udajov uzivatela';
            UsersVizu.StavyUsers_Index:= 9;
            IF UsersVizu.Edit_MenoUzivatela = '' OR UsersVizu.Edit_CisloKarty = '' THEN
                UsersVizu.StavyUsers_Index:= 13; //Zobrazenie stavov v textovom okne
                SC_Uzivatelia.ResetStep:= TRUE;
                SC_Uzivatelia.Step:= 0;
            ELSE
                SC_Uzivatelia.ResetStep:= TRUE;
                SC_Uzivatelia.Step:= 11;
            END_IF

        11://Kontrola mena už existujucich uzivatelov//
            SC_Uzivatelia.StepName:= '11 - Kontrola mena uz existujucich uzivatelov';
            IF Uzivatel[c].Meno = UsersVizu.Edit_MenoUzivatela THEN
                UsersVizu.StavyUsers_Index:= 2;
                SC_Uzivatelia.ResetStep:= TRUE;
                SC_Uzivatelia.Step:= 0;
            ELSE
                IF c < 100 THEN
                    c:= c + 1;
                ELSE
                    SC_Uzivatelia.ResetStep:= TRUE;
					SC_Uzivatelia.Step:= 12;
				END_IF
			END_IF

		12://Zistenie prázdneho pola pre uloženie receptury//
			SC_Uzivatelia.StepName:= '12 - Zistenie volneho pola';
			IF Uzivatel[d].Meno= '' THEN
				IndexPrazdPole:= d;
				SC_Uzivatelia.ResetStep:= TRUE;
				SC_Uzivatelia.Step:= 13;
			ELSE
				IF d < 100 THEN
					d:= d + 1;
				ELSE
					SC_Uzivatelia.ResetStep:= TRUE;
					SC_Uzivatelia.Step:= 0;
				END_IF
			END_IF

		13://Ulozenie uzivatela//
			SC_Uzivatelia.StepName:= '13 - Ulozenie uzivatela';
			Uzivatel[IndexPrazdPole].Meno:= UsersVizu.Edit_MenoUzivatela;
            Uzivatel[IndexPrazdPole].CisloKarty:= UsersVizu.Edit_CisloKarty;
            UrovenUzivatela:= STRING_TO_UINT(UsersVizu.Edit_UrovenUzivatela);
            Uzivatel[IndexPrazdPole].UrovenUzivatela:= UrovenUzivatela;
            MpRecipeXml_1.Save:= TRUE;
            IF MpRecipeXml_1.CommandDone THEN
                UsersVizu.StavyUsers_Index:= 1;
                UsersVizu.Edit_MenoUzivatela:= '';
                UsersVizu.Edit_CisloKarty:= '';
                SC_Uzivatelia.ResetStep:= TRUE;
                SC_Uzivatelia.Step:= 0;
		    END_IF

        20://Načítanie parametrov uživatela//
            SC_Uzivatelia.StepName:= '20 - Nacitanie parametrov uzivatela';
            UsersVizu.StavyUsers_Index:= 9;
            UsersVizu.Edit_MenoUzivatela:= Uzivatel[e].Meno;
            UsersVizu.Edit_HesloUzivatela:= Uzivatel[e].Heslo;
            UrovenUzivatela:= Uzivatel[e].UrovenUzivatela;
            UsersVizu.Edit_UrovenUzivatela:= UINT_TO_STRING(UrovenUzivatela);
            (*UsersVizu.Edit_CisloKarty:= Uzivatel[e].CisloKarty;*)
            UsersVizu.StavyUsers_Index:= 3;
            SC_Uzivatelia.ResetStep:= TRUE;
            SC_Uzivatelia.Step:= 0;

        30://Vymazanie uživatela//
            SC_Uzivatelia.StepName:= '30 - Vymazanie uzivatela';
            UsersVizu.StavyUsers_Index:= 9;
            Uzivatel[e].Meno:= '';
            Uzivatel[e].Heslo:= '';
            Uzivatel[e].CisloKarty:= '';
            Uzivatel[e].UrovenUzivatela:= 0;
            MpRecipeXml_1.Save:= TRUE;
            IF MpRecipeXml_1.CommandDone THEN
                UsersVizu.StavyUsers_Index:= 4;
                SC_Uzivatelia.ResetStep:= TRUE;
                SC_Uzivatelia.Step:= 0;
            END_IF

    END_CASE

				END_PROGRAM

PROGRAM _EXIT
				(* Insert code here *)

				END_PROGRAM
```

#### Variables.var - Local variables
```iecst
VAR
	strCategory : STRING[80];
	MpRecipeUI_1 : MpRecipeUI;
	UISetup : MpRecipeUISetupType;
	UIConnect : MpRecipeUIConnectType := (0);
	i : UINT := 0;
	a : UINT;
	CasOdhlaseniaUzivatela : TON;
	ListBoxPole_Sprava : ARRAY[0..100] OF STRING[100];
	ListBox_Value : ARRAY[0..100] OF STRING[10];
	b : USINT;
	c : UINT;
	IndexPrazdPole : UINT;
	d : UINT;
	e : UINT;
	f : UINT;
	g : UINT;
	h : UINT;
	SC_Uzivatelia : SequenceControlTyp;
	UrovenUzivatela : UINT;
END_VAR
```

### Program Logical/Uzivatelia/Users_Panel1 (IEC)

#### Main.st - Init, cyclic, exit code
```iecst
PROGRAM _INIT

END_PROGRAM

PROGRAM _CYCLIC

    //Volanie funkcie SequenceControl//
    SequenceControl(SC:= SC_Uzivatelia);

    //************************************Konvertovanie kódu čitačky do stringu****************************************************//
    FOR i:= 0 TO 7 BY 1 DO
        brsstrcpy(ADR(PrecitaneDataSTRING[i]),ADR(PrecitaneData_Panel1[i]));
    END_FOR

    //Spajanie pola stringov do stringu//
    KodCitackySTRING:= PrecitaneDataSTRING[0];
    brsstrcat(ADR(KodCitackySTRING), ADR(PrecitaneDataSTRING[1]));
    brsstrcat(ADR(KodCitackySTRING), ADR(PrecitaneDataSTRING[2]));
    brsstrcat(ADR(KodCitackySTRING), ADR(PrecitaneDataSTRING[3]));
    brsstrcat(ADR(KodCitackySTRING), ADR(PrecitaneDataSTRING[4]));
    brsstrcat(ADR(KodCitackySTRING), ADR(PrecitaneDataSTRING[5]));
    brsstrcat(ADR(KodCitackySTRING), ADR(PrecitaneDataSTRING[6]));
    brsstrcat(ADR(KodCitackySTRING), ADR(PrecitaneDataSTRING[7]));

    IF KodCitackySTRING = '' THEN
        CisloPrihlasenejKarty_Panel1:= '';
    ELSE
        CisloPrihlasenejKarty_Panel1:= KodCitackySTRING;
    END_IF

    //**************************************************Kontrola či je karta priložená******************************************************//

    IF KodCitackySTRING <> '' THEN
        CasControlyKarty.IN:= TRUE;
    ELSE
        CasControlyKarty.IN:= FALSE;
    END_IF

    IF CasControlyKarty.Q THEN
        UsersVizu.KartaPrilozena_Panel1:= TRUE;
    ELSE
        UsersVizu.KartaPrilozena_Panel1:= FALSE;
    END_IF

    CasControlyKarty.PT:= T#1s;
    CasControlyKarty();

    //***************************************************Kontrola či je uživatel už prihlásený**********************************************//
    IF UsersVizu.MenoPrihlasenehoUzivatela_Panel1 = '' THEN
        P1_UzivatelPrihlaseny:= FALSE;
    ELSE
        P1_UzivatelPrihlaseny:= TRUE;
    END_IF
//    P1_UzivatelPrihlaseny:= TRUE;
//    P1_UrovenPrihlasenehoUzivatela:= 20;

    //Kontrola karty//

    IF KodCitackySTRING = '' THEN
        PrecitaneCisloKarty:= '';
    ELSE
        PrecitaneCisloKarty:= KodCitackySTRING;
    END_IF

    CASE SC_Uzivatelia.Step OF

        0://Nulovanie//
            SC_Uzivatelia.StepName:= '0 - Nulovanie';
            UsersVizu.OdhlasUzivatela_Panel1:= FALSE;
            a:= 0;
            SC_Uzivatelia.ResetStep:= TRUE;
            SC_Uzivatelia.Step:= 1;

        1://Rozhodnutie o činnosti//
            SC_Uzivatelia.StepName:= '1 - Rozhodnutie o cinnosti';
            IF UsersVizu.KartaPrilozena_Panel1 AND P1_Vizu.ActualPage <> 'PageUsers' THEN
                SC_Uzivatelia.ResetStep:= TRUE;
                SC_Uzivatelia.Step:= 10;
            ELSIF UsersVizu.OdhlasUzivatela_Panel1 THEN
                SC_Uzivatelia.ResetStep:= TRUE;
                SC_Uzivatelia.Step:= 20;
            END_IF

        10://Kontrola udajov karty//
            SC_Uzivatelia.StepName:= '10 - Kontrola udajov karty';
            SC_Uzivatelia.IdleTime.PT:= T#2s;
            SC_Uzivatelia.AlarmTime.PT:= T#2s;

            IF NOT P1_UzivatelPrihlaseny THEN
                IF PrecitaneCisloKarty <> '' THEN
                    SC_Uzivatelia.ResetStep:= TRUE;
                    SC_Uzivatelia.Step:= 13;
                ELSE
                    SC_Uzivatelia.ResetStep:= TRUE;
                    SC_Uzivatelia.Step:= 100;
                END_IF
            ELSE
                SC_Uzivatelia.ResetStep:= TRUE;
                SC_Uzivatelia.Step:= 100;
            END_IF

        13://Hladanie prihlaseného uživatela v zoznamoch//
            SC_Uzivatelia.StepName:= '13 - Hladanie prihlaseneho uzivatela';
            SC_Uzivatelia.IdleTime.PT:= T#2s;
            SC_Uzivatelia.AlarmTime.PT:= T#2s;

            IF Uzivatel[a].CisloKarty = PrecitaneCisloKarty THEN
                UsersVizu.MenoPrihlasenehoUzivatela_Panel1:= Uzivatel[a].Meno;
                UsersVizu.CisloPrihlasenejKarty_Panel1:= Uzivatel[a].CisloKarty;
                P1_UrovenPrihlasenehoUzivatela:= Uzivatel[a].UrovenUzivatela;
                SC_Uzivatelia.ResetStep:= TRUE;
                SC_Uzivatelia.Step:= 100;
            ELSE
                IF a < 100 THEN
                    a:= a + 1;
                ELSE
                    SC_Uzivatelia.ResetStep:= TRUE;
                    SC_Uzivatelia.Step:= 15;
                END_IF
            END_IF

        15://Priradenie čísla karty//
            SC_Uzivatelia.StepName:= '15 - Priradenie cisla karty';
            SC_Uzivatelia.IdleTime.PT:= T#2s;
            SC_Uzivatelia.AlarmTime.PT:= T#2s;

            UsersVizu.MenoPrihlasenehoUzivatela_Panel1:= 'Operator';
            UsersVizu.CisloPrihlasenejKarty_Panel1:= PrecitaneCisloKarty;
            SC_Uzivatelia.ResetStep:= TRUE;
            SC_Uzivatelia.Step:= 100;

        20://Odhlásenie uživatela//
            SC_Uzivatelia.StepName:= '20 - Odhlasenie uzivatela';
            SC_Uzivatelia.IdleTime.PT:= T#2s;
            SC_Uzivatelia.AlarmTime.PT:= T#2s;

            UsersVizu.MenoPrihlasenehoUzivatela_Panel1:= '';
            UsersVizu.CisloPrihlasenejKarty_Panel1:= '';
            P1_UrovenPrihlasenehoUzivatela:= 0;
            SC_Uzivatelia.ResetStep:= TRUE;
            SC_Uzivatelia.Step:= 100;

        100://Čakam na odobratie karty//
            SC_Uzivatelia.StepName:= '110 - Cakanie na odobratie karty';
            SC_Uzivatelia.IdleTime.PT:= T#1s;
            SC_Uzivatelia.AlarmTime.PT:= T#2s;

            SC_Uzivatelia.IdleTime.IN:= NOT UsersVizu.KartaPrilozena_Panel1;

            IF SC_Uzivatelia.IdleTime.Q THEN
                SC_Uzivatelia.ResetStep:= TRUE;
                SC_Uzivatelia.Step:= 0;
            END_IF

    END_CASE

END_PROGRAM

PROGRAM _EXIT
	(* Insert code here *)

END_PROGRAM
```

#### Variables.var - Local variables
```iecst
VAR
	i : USINT;
	PrecitaneDataSTRING : ARRAY[0..7] OF STRING[1] := [8('')];
	KodCitackySTRING : STRING[80];
	CasControlyKarty : TON;
	SC_Uzivatelia : SequenceControlTyp;
	PrecitaneCisloKarty : STRING[80];
	a : USINT;
END_VAR
```

### Program Logical/Uzivatelia/Users_Panel2 (IEC)

#### Main.st - Init, cyclic, exit code
```iecst
PROGRAM _INIT

END_PROGRAM

PROGRAM _CYCLIC

    //Volanie funkcie SequenceControl//
    SequenceControl(SC:= SC_Uzivatelia);

    //************************************Konvertovanie kódu čitačky do stringu****************************************************//
    FOR i:= 0 TO 7 BY 1 DO
        brsstrcpy(ADR(PrecitaneDataSTRING[i]),ADR(PrecitaneData_Panel2[i]));
    END_FOR

    //Spajanie pola stringov do stringu//
    KodCitackySTRING:= PrecitaneDataSTRING[0];
    brsstrcat(ADR(KodCitackySTRING), ADR(PrecitaneDataSTRING[1]));
    brsstrcat(ADR(KodCitackySTRING), ADR(PrecitaneDataSTRING[2]));
    brsstrcat(ADR(KodCitackySTRING), ADR(PrecitaneDataSTRING[3]));
    brsstrcat(ADR(KodCitackySTRING), ADR(PrecitaneDataSTRING[4]));
    brsstrcat(ADR(KodCitackySTRING), ADR(PrecitaneDataSTRING[5]));
    brsstrcat(ADR(KodCitackySTRING), ADR(PrecitaneDataSTRING[6]));
    brsstrcat(ADR(KodCitackySTRING), ADR(PrecitaneDataSTRING[7]));

    //**************************************************Kontrola či je karta priložená******************************************************//

    IF KodCitackySTRING <> '' THEN
        CasControlyKarty.IN:= TRUE;
    ELSE
        CasControlyKarty.IN:= FALSE;
    END_IF

    IF CasControlyKarty.Q THEN
        UsersVizu.KartaPrilozena_Panel2:= TRUE;
    ELSE
        UsersVizu.KartaPrilozena_Panel2:= FALSE;
    END_IF

    CasControlyKarty.PT:= T#1s;
    CasControlyKarty();

    //***************************************************Kontrola či je uživatel už prihlásený**********************************************//
    IF UsersVizu.MenoPrihlasenehoUzivatela_Panel2 = '' THEN
        P2_UzivatelPrihlaseny:= FALSE;
    ELSE
        P2_UzivatelPrihlaseny:= TRUE;
    END_IF

//    P2_UzivatelPrihlaseny:= TRUE;
//    P2_UrovenPrihlasenehoUzivatela:= 20;

    //Kontrola karty//

    IF KodCitackySTRING = '' THEN
        PrecitaneCisloKarty:= '';
    ELSE
        PrecitaneCisloKarty:= KodCitackySTRING;
    END_IF

    CASE SC_Uzivatelia.Step OF

        0://Nulovanie//
            SC_Uzivatelia.StepName:= '0 - Nulovanie';
            UsersVizu.OdhlasUzivatela_Panel2:= FALSE;
            a:= 0;
            SC_Uzivatelia.ResetStep:= TRUE;
            SC_Uzivatelia.Step:= 1;

        1://Rozhodnutie o činnosti//
            SC_Uzivatelia.StepName:= '1 - Rozhodnutie o cinnosti';
            IF UsersVizu.KartaPrilozena_Panel2 THEN
                SC_Uzivatelia.ResetStep:= TRUE;
                SC_Uzivatelia.Step:= 10;
            ELSIF UsersVizu.OdhlasUzivatela_Panel2 THEN
                SC_Uzivatelia.ResetStep:= TRUE;
                SC_Uzivatelia.Step:= 20;
            END_IF

        10://Kontrola udajov karty//
            SC_Uzivatelia.StepName:= '10 - Kontrola udajov karty';
            SC_Uzivatelia.IdleTime.PT:= T#2s;
            SC_Uzivatelia.AlarmTime.PT:= T#2s;

            IF NOT P2_UzivatelPrihlaseny THEN
                IF PrecitaneCisloKarty <> '' THEN
                    SC_Uzivatelia.ResetStep:= TRUE;
                    SC_Uzivatelia.Step:= 13;
                ELSE
                    SC_Uzivatelia.ResetStep:= TRUE;
                    SC_Uzivatelia.Step:= 100;
                END_IF
            ELSE
                SC_Uzivatelia.ResetStep:= TRUE;
                SC_Uzivatelia.Step:= 100;
            END_IF

        13://Hladanie prihlaseného uživatela v zoznamoch//
            SC_Uzivatelia.StepName:= '13 - Hladanie prihlaseneho uzivatela';
            SC_Uzivatelia.IdleTime.PT:= T#2s;
            SC_Uzivatelia.AlarmTime.PT:= T#2s;

            IF Uzivatel[a].CisloKarty = PrecitaneCisloKarty THEN
                UsersVizu.MenoPrihlasenehoUzivatela_Panel2:= Uzivatel[a].Meno;
                UsersVizu.CisloPrihlasenejKarty_Panel2:= Uzivatel[a].CisloKarty;
                P2_UrovenPrihlasenehoUzivatela:= Uzivatel[a].UrovenUzivatela;
                SC_Uzivatelia.ResetStep:= TRUE;
                SC_Uzivatelia.Step:= 100;
            ELSE
                IF a < 100 THEN
                    a:= a + 1;
                ELSE
                    SC_Uzivatelia.ResetStep:= TRUE;
                    SC_Uzivatelia.Step:= 15;
                END_IF
            END_IF

        15://Priradenie čísla karty//
            SC_Uzivatelia.StepName:= '15 - Priradenie cisla karty';
            SC_Uzivatelia.IdleTime.PT:= T#2s;
            SC_Uzivatelia.AlarmTime.PT:= T#2s;

            UsersVizu.MenoPrihlasenehoUzivatela_Panel2:= 'Operator';
            UsersVizu.CisloPrihlasenejKarty_Panel2:= PrecitaneCisloKarty;
            SC_Uzivatelia.ResetStep:= TRUE;
            SC_Uzivatelia.Step:= 100;

        20://Odhlásenie uživatela//
            SC_Uzivatelia.StepName:= '20 - Odhlasenie uzivatela';
            SC_Uzivatelia.IdleTime.PT:= T#2s;
            SC_Uzivatelia.AlarmTime.PT:= T#2s;

            UsersVizu.MenoPrihlasenehoUzivatela_Panel2:= '';
            UsersVizu.CisloPrihlasenejKarty_Panel2:= '';
            P2_UrovenPrihlasenehoUzivatela:= 0;
            SC_Uzivatelia.ResetStep:= TRUE;
            SC_Uzivatelia.Step:= 100;

        100://Čakam na odobratie karty//
            SC_Uzivatelia.StepName:= '110 - Cakanie na odobratie karty';
            SC_Uzivatelia.IdleTime.PT:= T#1s;
            SC_Uzivatelia.AlarmTime.PT:= T#2s;

            SC_Uzivatelia.IdleTime.IN:= NOT UsersVizu.KartaPrilozena_Panel2;

            IF SC_Uzivatelia.IdleTime.Q THEN
                SC_Uzivatelia.ResetStep:= TRUE;
                SC_Uzivatelia.Step:= 0;
            END_IF

    END_CASE

END_PROGRAM

PROGRAM _EXIT
	(* Insert code here *)

END_PROGRAM
```

#### Variables.var - Local variables
```iecst
VAR
	i : USINT;
	PrecitaneDataSTRING : ARRAY[0..7] OF STRING[1] := [8('')];
	KodCitackySTRING : STRING[80];
	CasControlyKarty : TON;
	SC_Uzivatelia : SequenceControlTyp;
	PrecitaneCisloKarty : STRING[80];
	a : USINT;
END_VAR
```

### Program Logical/Uzivatelia/Users_Panel3 (IEC)

#### Main.st - Init, cyclic, exit code
```iecst
PROGRAM _INIT

END_PROGRAM

PROGRAM _CYCLIC

    //Volanie funkcie SequenceControl//
    SequenceControl(SC:= SC_Uzivatelia);

      //************************************Konvertovanie kódu čitačky do stringu****************************************************//
    FOR i:= 0 TO 7 BY 1 DO
        brsstrcpy(ADR(PrecitaneDataSTRING[i]),ADR(PrecitaneData_Panel3[i]));
    END_FOR

    //Spajanie pola stringov do stringu//
    KodCitackySTRING:= PrecitaneDataSTRING[0];
    brsstrcat(ADR(KodCitackySTRING), ADR(PrecitaneDataSTRING[1]));
    brsstrcat(ADR(KodCitackySTRING), ADR(PrecitaneDataSTRING[2]));
    brsstrcat(ADR(KodCitackySTRING), ADR(PrecitaneDataSTRING[3]));
    brsstrcat(ADR(KodCitackySTRING), ADR(PrecitaneDataSTRING[4]));
    brsstrcat(ADR(KodCitackySTRING), ADR(PrecitaneDataSTRING[5]));
    brsstrcat(ADR(KodCitackySTRING), ADR(PrecitaneDataSTRING[6]));
    brsstrcat(ADR(KodCitackySTRING), ADR(PrecitaneDataSTRING[7]));

    //**************************************************Kontrola či je karta priložená******************************************************//

    IF KodCitackySTRING <> '' THEN
        CasControlyKarty.IN:= TRUE;
    ELSE
        CasControlyKarty.IN:= FALSE;
    END_IF

    IF CasControlyKarty.Q THEN
        UsersVizu.KartaPrilozena_Panel3:= TRUE;
    ELSE
        UsersVizu.KartaPrilozena_Panel3:= FALSE;
    END_IF

    CasControlyKarty.PT:= T#1s;
    CasControlyKarty();

    //***************************************************Kontrola či je uživatel už prihlásený**********************************************//
    IF UsersVizu.MenoPrihlasenehoUzivatela_Panel3 = '' THEN
        P34_UzivatelPrihlaseny:= FALSE;
    ELSE
        P34_UzivatelPrihlaseny:= TRUE;
    END_IF

//    P34_UzivatelPrihlaseny:= TRUE;
//    P34_UrovenPrihlasenehoUzivatela:= 20;

    //Kontrola karty//

    IF KodCitackySTRING = '' THEN
        PrecitaneCisloKarty:= '';
    ELSE
        PrecitaneCisloKarty:= KodCitackySTRING;
    END_IF

    CASE SC_Uzivatelia.Step OF

        0://Nulovanie//
            SC_Uzivatelia.StepName:= '0 - Nulovanie';
            UsersVizu.OdhlasUzivatela_Panel3:= FALSE;
            a:= 0;
            SC_Uzivatelia.ResetStep:= TRUE;
            SC_Uzivatelia.Step:= 1;

        1://Rozhodnutie o činnosti//
            SC_Uzivatelia.StepName:= '1 - Rozhodnutie o cinnosti';
            IF UsersVizu.KartaPrilozena_Panel3 THEN
                SC_Uzivatelia.ResetStep:= TRUE;
                SC_Uzivatelia.Step:= 10;
            ELSIF UsersVizu.OdhlasUzivatela_Panel3 THEN
                SC_Uzivatelia.ResetStep:= TRUE;
                SC_Uzivatelia.Step:= 20;
            END_IF

        10://Kontrola udajov karty//
            SC_Uzivatelia.StepName:= '10 - Kontrola udajov karty';
            SC_Uzivatelia.IdleTime.PT:= T#2s;
            SC_Uzivatelia.AlarmTime.PT:= T#2s;

            IF NOT P34_UzivatelPrihlaseny THEN
                IF PrecitaneCisloKarty <> '' THEN
                    SC_Uzivatelia.ResetStep:= TRUE;
                    SC_Uzivatelia.Step:= 13;
                ELSE
                    SC_Uzivatelia.ResetStep:= TRUE;
                    SC_Uzivatelia.Step:= 100;
                END_IF
            ELSE
                SC_Uzivatelia.ResetStep:= TRUE;
                SC_Uzivatelia.Step:= 100;
            END_IF

        13://Hladanie prihlaseného uživatela v zoznamoch//
            SC_Uzivatelia.StepName:= '13 - Hladanie prihlaseneho uzivatela';
            SC_Uzivatelia.IdleTime.PT:= T#2s;
            SC_Uzivatelia.AlarmTime.PT:= T#2s;

            IF Uzivatel[a].CisloKarty = PrecitaneCisloKarty THEN
                UsersVizu.MenoPrihlasenehoUzivatela_Panel3:= Uzivatel[a].Meno;
                UsersVizu.CisloPrihlasenejKarty_Panel3:= Uzivatel[a].CisloKarty;
                P34_UrovenPrihlasenehoUzivatela:= Uzivatel[a].UrovenUzivatela;
                SC_Uzivatelia.ResetStep:= TRUE;
                SC_Uzivatelia.Step:= 100;
            ELSE
                IF a < 100 THEN
                    a:= a + 1;
                ELSE
                    SC_Uzivatelia.ResetStep:= TRUE;
                    SC_Uzivatelia.Step:= 15;
                END_IF
            END_IF

        15://Priradenie čísla karty//
            SC_Uzivatelia.StepName:= '15 - Priradenie cisla karty';
            SC_Uzivatelia.IdleTime.PT:= T#2s;
            SC_Uzivatelia.AlarmTime.PT:= T#2s;

            UsersVizu.MenoPrihlasenehoUzivatela_Panel3:= 'Operator';
            UsersVizu.CisloPrihlasenejKarty_Panel1:= PrecitaneCisloKarty;
            SC_Uzivatelia.ResetStep:= TRUE;
            SC_Uzivatelia.Step:= 100;

        20://Odhlásenie uživatela//
            SC_Uzivatelia.StepName:= '20 - Odhlasenie uzivatela';
            SC_Uzivatelia.IdleTime.PT:= T#2s;
            SC_Uzivatelia.AlarmTime.PT:= T#2s;

            UsersVizu.MenoPrihlasenehoUzivatela_Panel3:= '';
            UsersVizu.CisloPrihlasenejKarty_Panel3:= '';
            P34_UrovenPrihlasenehoUzivatela:= 0;
            SC_Uzivatelia.ResetStep:= TRUE;
            SC_Uzivatelia.Step:= 100;

        100://Čakam na odobratie karty//
            SC_Uzivatelia.StepName:= '110 - Cakanie na odobratie karty';
            SC_Uzivatelia.IdleTime.PT:= T#1s;
            SC_Uzivatelia.AlarmTime.PT:= T#2s;

            SC_Uzivatelia.IdleTime.IN:= NOT UsersVizu.KartaPrilozena_Panel3;

            IF SC_Uzivatelia.IdleTime.Q THEN
                SC_Uzivatelia.ResetStep:= TRUE;
                SC_Uzivatelia.Step:= 0;
            END_IF

    END_CASE

END_PROGRAM

PROGRAM _EXIT
	(* Insert code here *)

END_PROGRAM
```

#### Variables.var - Local variables
```iecst
VAR
	i : USINT;
	PrecitaneDataSTRING : ARRAY[0..7] OF STRING[1] := [8('')];
	KodCitackySTRING : STRING[80];
	CasControlyKarty : TON;
	SC_Uzivatelia : SequenceControlTyp;
	PrecitaneCisloKarty : STRING[80];
	a : USINT;
END_VAR
```

### DatumCasGlobal.var
```iecst
VAR
	PLC_Cas : PLC_Cas_typ;
	PLC_Datum : PLC_Datum_typ;
	Sekunda_STR : STRING[2];
	Minuta_STR : STRING[2];
	Hodina_STR : STRING[2];
	Den_STR : STRING[2];
	Mesiac_STR : STRING[2];
	Rok_STR_4_Znaky : STRING[4];
	Rok_STR_2_Znaky : STRING[2];
END_VAR
```

### DatumCasGlobal.typ
```iecst
TYPE
	PLC_Cas_typ : 	STRUCT
		Sekundy : USINT;
		Minuty : USINT;
		Hodiny : USINT;
	END_STRUCT;
	PLC_Datum_typ : 	STRUCT
		Den : USINT;
		Mesiac : USINT;
		Rok : UINT;
	END_STRUCT;
END_TYPE
```

### Program Logical/DatumCasPLC/DatumCasPLC (IEC)

#### Main.st - Init, cyclic, exit code
```iecst
PROGRAM _INIT
	(* Insert code here *)

END_PROGRAM

PROGRAM _CYCLIC

	//Vyčítavanie systémového času//
	DTGetTime_1.enable:= TRUE;
	DTGetTime_1();
	DT_TO_DTStructure(DTGetTime_1.DT1,ADR(PLC_DatumCas));

	PLC_Cas.Sekundy:= PLC_DatumCas.second;
	PLC_Cas.Minuty:= PLC_DatumCas.minute;
	PLC_Cas.Hodiny:= PLC_DatumCas.hour;

	PLC_Datum.Den:= PLC_DatumCas.day;
	PLC_Datum.Mesiac:= PLC_DatumCas.month;
	PLC_Datum.Rok:= PLC_DatumCas.year;

	//Prevod času na String//
	//Sekundy//
	IF PLC_Cas.Sekundy < 10 THEN
		Sekundy_String:= USINT_TO_STRING(PLC_Cas.Sekundy);
		Sekunda_STR:= '0';
		brsstrcat(ADR(Sekunda_STR),ADR(Sekundy_String));
	ELSE
		Sekunda_STR:= USINT_TO_STRING(PLC_Cas.Sekundy);
	END_IF

	//Minuty//
	IF PLC_Cas.Minuty < 10 THEN
		Minuty_String:= USINT_TO_STRING(PLC_Cas.Minuty);
		Minuta_STR:= '0';
		brsstrcat(ADR(Minuta_STR),ADR(Minuty_String));
	ELSE
		Minuta_STR:= USINT_TO_STRING(PLC_Cas.Minuty);
	END_IF

	//Hodiny//
	IF PLC_Cas.Hodiny < 10 THEN
		Hodiny_String:= USINT_TO_STRING(PLC_Cas.Hodiny);
		Hodina_STR:= '0';
		brsstrcat(ADR(Hodina_STR),ADR(Hodiny_String));
	ELSE
		Hodina_STR:= USINT_TO_STRING(PLC_Cas.Hodiny);
	END_IF

	//Prevod dátumu na String//
	//Deň//
	IF PLC_Datum.Den < 10 THEN
		Den_String:= USINT_TO_STRING(PLC_Datum.Den);
		Den_STR:= '0';
		brsstrcat(ADR(Den_STR),ADR(Den_String));
	ELSE
		Den_STR:= USINT_TO_STRING(PLC_Datum.Den);
	END_IF

	//Masiac//
	IF PLC_Datum.Mesiac < 10 THEN
		Mesiac_String:= USINT_TO_STRING(PLC_Datum.Mesiac);
		Mesiac_STR:= '0';
		brsstrcat(ADR(Mesiac_STR),ADR(Mesiac_String));
	ELSE
		Mesiac_STR:= USINT_TO_STRING(PLC_Datum.Mesiac);
	END_IF

	//Rok - 4 znaky//
	Rok_STR_4_Znaky:= UINT_TO_STRING(PLC_Datum.Rok);

	//Rok - posledné 2 znaky//
	length := brsstrlen(ADR(Rok_STR_4_Znaky)); //Zistí počet znakov//

	IF length >= 4 THEN
		brsmemcpy(ADR(PoleUSINT),ADR(Rok_STR_4_Znaky),SIZEOF(Rok_STR_4_Znaky));
		i := PoleUSINT[length-2]; //Vyčítanie predposledného znaku//
		brsstrcpy(ADR(DvaZnaky),ADR(i));
		i := PoleUSINT[length-1]; //Vyčítanie posledneho znaku//
		brsstrcat(ADR(DvaZnaky),ADR(i));
	END_IF

	Rok_STR_2_Znaky:= DvaZnaky;

END_PROGRAM

PROGRAM _EXIT
	(* Insert code here *)

END_PROGRAM
```

#### Variables.var - Local variables
```iecst
VAR
	PLC_DatumCas : DTStructure;
	DTGetTime_1 : DTGetTime;
	Sekundy_String : STRING[2];
	Minuty_String : STRING[2];
	Hodiny_String : STRING[2];
	Den_String : STRING[2];
	Mesiac_String : STRING[2];
	length : UDINT;
	PoleUSINT : ARRAY[0..3] OF USINT;
	i : USINT;
	DvaZnaky : STRING[2];
END_VAR
```

### Poznamky.txt
```
Prihlasovacie údaje na FTP:
Login - admin
Heslo - vlmardo

Prihlasovacie údaje do Safety:
Heslo - vlmardo

//*********APC Windows*************//
Heslo - vlmardoDMP

//**********Vzdialená plocha**********//
192.168.122.3
Meno - remote
Heslo - vlmardo

//***********Prístup na FTP SSD disk PLC*******//
IP 192.168.122.3
Meno - remote
Heslo - vlmardo

//************Prístup na FTP kameru č.1 na disku PLC*********//
IP 192.168.122.4
Meno - cam1
Heslo - .cam1

//************Prístup na FTP Panasonic*******************//
IP 192.168.100.164
Meno - designMP
Heslo - Ftp4PAN2020

Pre spojenie je potrebné vypnúť wifi

**********Pracovisko 1*************
Výťah:
- Servo zdvihu výťahu - prevod 5mm/ot
Šrobovanie:
- Servo manipulatora Os X - prevod 10mm/ot
- Servo manipulatora Os Y - prevod 10mm/ot

***********Pracovisko 2*************
Zakladač izolácie:
- Servo zdvihu - prevod 10mm/ot  Celkový zdvih 100mm
- Servo pojazdu vozíka - prevod 132mm/ot
Šrobovanie:
- Servo manipulatora Os X - prevod 10mm/ot
- Servo manipulatora Os Y - prevod 10mm/ot
Zváranie:
- Servo zdvihu zvárania - prevod 10mm/ot Celkový zdvih 310mm

*****************Číslovanie kamier*************************
CAM 1 - Control Unit CAM 4
CAM 2 - Control Unit CAM 1
CAM 4 - Control Unit CAM 2
CAM 6 - Control Unit CAM 3
CAM 7 - Control Unit CAM 5
CAM 10 - Control Unit CAM 7
CAM 11 - Control Unit CAM 8
CAM 12 - Control Unit CAM 9
CAM 15 - Control Unit CAM 10
CAM 16 - Control Unit CAM 11
CAM 17 - Control Unit CAM 6

CAM 9 - Smart kamera CAM9
IP kamerového systému 192.168.148.30
Heslo - vision

**************************Postup kalibrácie vysunutia šróbovačiek***********************************
- na pracovisku zacentrujeme paletku

********P1 Skrutkovanie*************
Skrutkovačka K30 - dištanc 60mm  východzia poloha
                 - opretie o paletku  koncová poloha

Skrutkovačka M5 - dištanc 60mm východzia poloha
                - opretie o paletku koncová poloha

Skrutkovačka M4 - dištanc 60mm východzia poloha
                - dištanc 12mm koncová poloha

*******P2 Maticovačka***************
Skrutkovačka matice M4 - dištanc 52mm východzia poloha
                       - dištanc 12mm koncová poloha

*******P2 Skrutkovanie****************
Skrutkovačka M6 - dištanc 72mm východzia poloha
                - dištanc 15mm koncová poloha

Skrutkovačka M4 - dištanc 87mm východzia poloha
                - dištanc 27mm koncová poloha

Skrutkovačka M5 - dištanc 115 mm východzia poloha
                - max vysunutie skrutkovačky koncová poloha

*******P3 Skrutkovanie******************
Skrutkovačka K40 - dištanc 52,5mm východzia poloha
                 - opretie o paletku  koncová poloha

Skrutkovačka M5 - dištanc 60mm  východzia poloha
                - opretie o paletku  koncová poloha

*****************************************************Kalibračné hodnoty skrutkovačiek***********************************************************
/Model 5H/

Srutkovanie 1:
Lavá K30 - 44.6 až 44.9
Pravá K30 - 44.5 až 44.8
Lavá M5 - 31.3 až 31.7
Pravá M5 - 31.0 až 31.5
Stredná M5 - 31.4 až 31.8

Skrutkovanie matice:
Vysunutie skrutkovačky - 37.5 až 37.8

Skrutkovanie 2:
Lavá M5 - 40.7 až 41.1
Pravá M5 - 40.7 až 41.0
Stredná M4 - 15.8 až 16.3

Skrutkovanie 3:
Stredná M5 - 42.0 až 42.3
```
